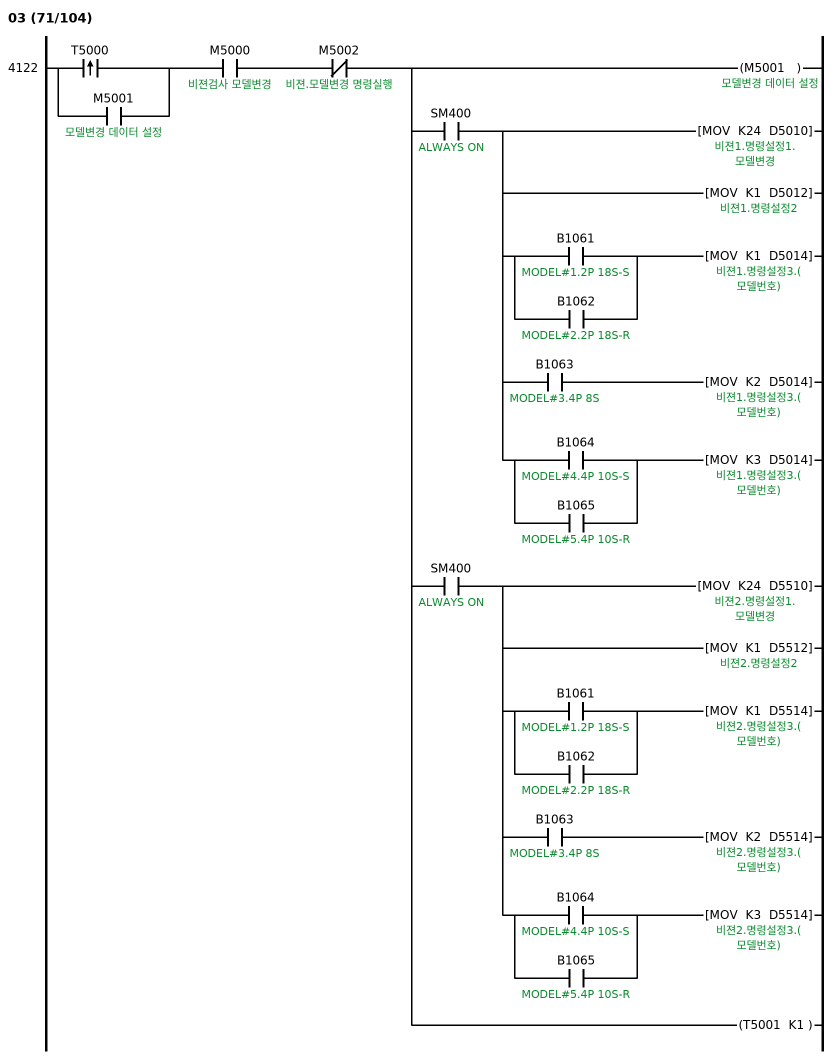
4122  LDP     T5000
      OR      M5001  ; 모델변경 데이터 설정
      AND     M5000  ; 비젼검사 모델변경
      ANI     M5002  ; 비젼.모델변경 명령실행
      OUT     M5001  ; 모델변경 데이터 설정
      MPS
      AND     SM400  ; ALWAYS ON
      MOV     K24 D5010  ; 비젼1.명령설정1.모델변경
      MOV     K1 D5012  ; 비젼1.명령설정2
      MPS
      LD      B1061  ; MODEL#1.2P 18S-S
      OR      B1062  ; MODEL#2.2P 18S-R
      ANB
      MOV     K1 D5014  ; 비젼1.명령설정3.(모델번호)
      MRD
      AND     B1063  ; MODEL#3.4P 8S
      MOV     K2 D5014
      MPP
      LD      B1064  ; MODEL#4.4P 10S-S
      OR      B1065  ; MODEL#5.4P 10S-R
      ANB
      MOV     K3 D5014
      MRD
      AND     SM400  ; ALWAYS ON
      MOV     K24 D5510  ; 비젼2.명령설정1.모델변경
      MOV     K1 D5512  ; 비젼2.명령설정2
      MPS
      LD      B1061  ; MODEL#1.2P 18S-S
      OR      B1062  ; MODEL#2.2P 18S-R
      ANB
      MOV     K1 D5514  ; 비젼2.명령설정3.(모델번호)
      MRD
      AND     B1063  ; MODEL#3.4P 8S
      MOV     K2 D5514
      MPP
      LD      B1064  ; MODEL#4.4P 10S-S
      OR      B1065  ; MODEL#5.4P 10S-R
      ANB
      MOV     K3 D5514
      MPP
      OUT     T5001 K1
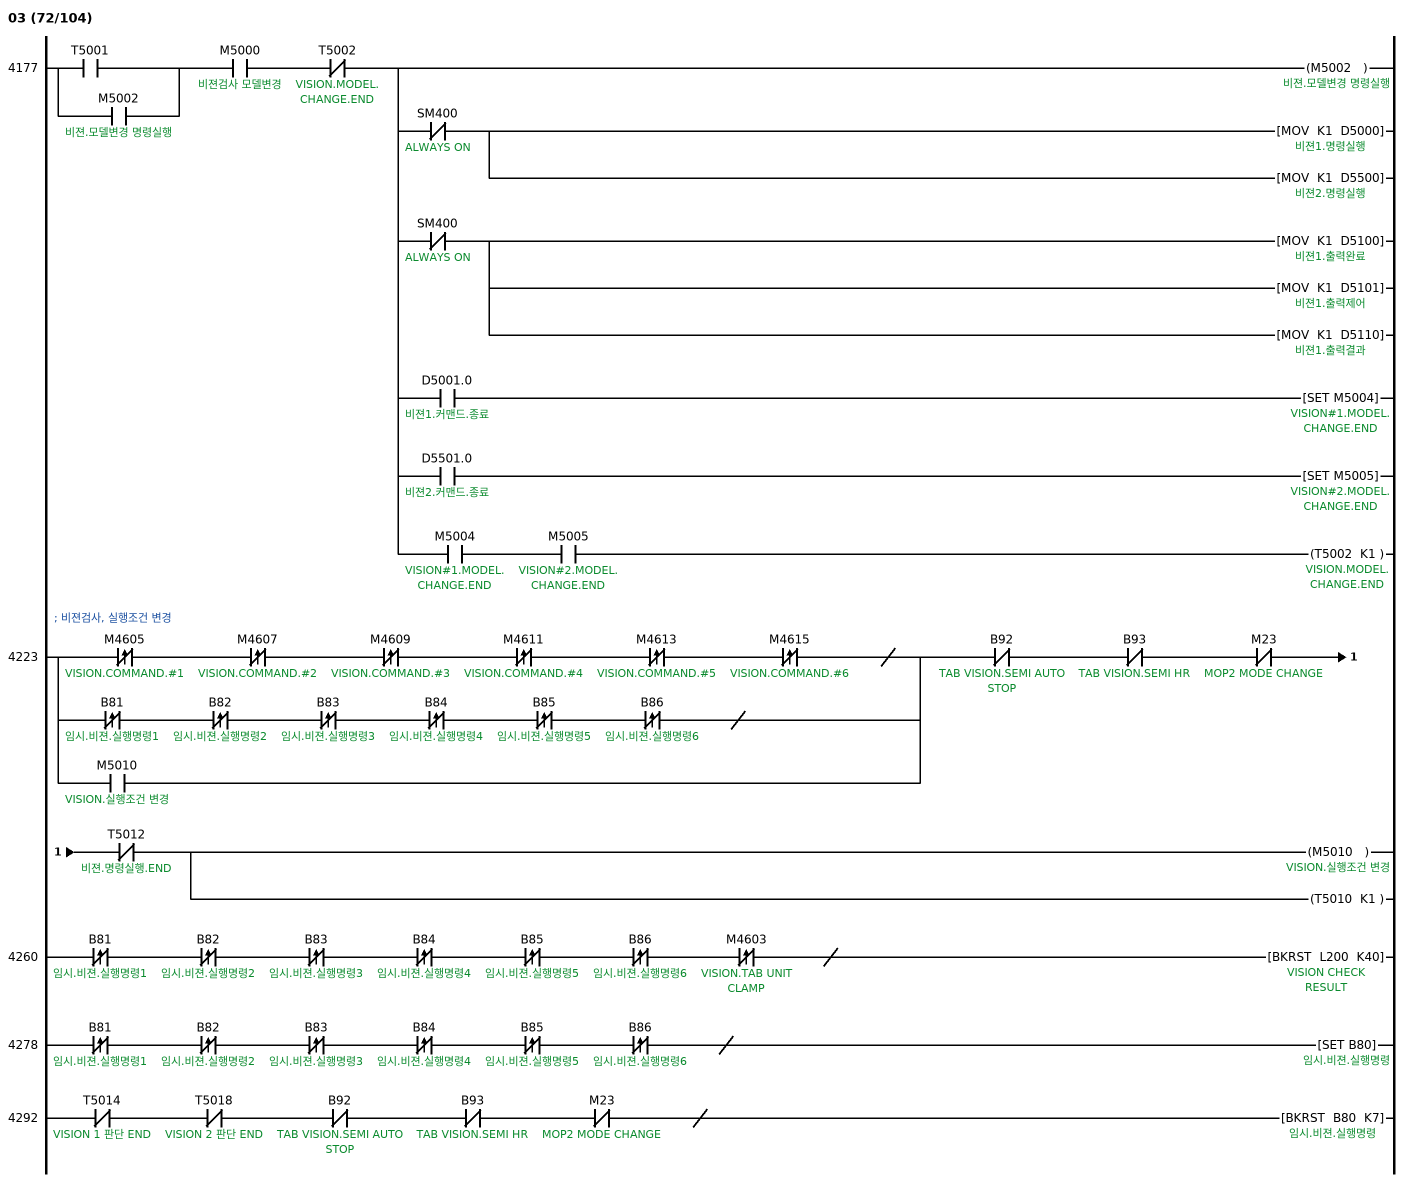
4177  LD      T5001
      OR      M5002  ; 비젼.모델변경 명령실행
      AND     M5000  ; 비젼검사 모델변경
      ANI     T5002  ; VISION.MODEL.CHANGE.END
      OUT     M5002  ; 비젼.모델변경 명령실행
      MPS
      ANI     SM400  ; ALWAYS ON
      MOV     K1 D5000  ; 비젼1.명령실행
      MOV     K1 D5500  ; 비젼2.명령실행
      MRD
      ANI     SM400  ; ALWAYS ON
      MOV     K1 D5100  ; 비젼1.출력완료
      MOV     K1 D5101  ; 비젼1.출력제어
      MOV     K1 D5110  ; 비젼1.출력결과
      MRD
      AND     D5001.0  ; 비젼1.커맨드.종료
      SET     M5004  ; VISION#1.MODEL.CHANGE.END
      MRD
      AND     D5501.0  ; 비젼2.커맨드.종료
      SET     M5005  ; VISION#2.MODEL.CHANGE.END
      MPP
      AND     M5004  ; VISION#1.MODEL.CHANGE.END
      AND     M5005  ; VISION#2.MODEL.CHANGE.END
      OUT     T5002 K1  ; VISION.MODEL.CHANGE.END
; 비젼검사, 실행조건 변경
4223  LDPI    M4605  ; VISION.COMMAND.#1
      ANDPI   M4607  ; VISION.COMMAND.#2
      ANDPI   M4609  ; VISION.COMMAND.#3
      ANDPI   M4611  ; VISION.COMMAND.#4
      ANDPI   M4613  ; VISION.COMMAND.#5
      ANDPI   M4615  ; VISION.COMMAND.#6
      INV
      LDPI    B81  ; 임시.비젼.실행명령1
      ANDPI   B82  ; 임시.비젼.실행명령2
      ANDPI   B83  ; 임시.비젼.실행명령3
      ANDPI   B84  ; 임시.비젼.실행명령4
      ANDPI   B85  ; 임시.비젼.실행명령5
      ANDPI   B86  ; 임시.비젼.실행명령6
      INV
      ORB
      OR      M5010  ; VISION.실행조건 변경
      ANI     B92  ; TAB VISION.SEMI AUTO STOP
      ANI     B93  ; TAB VISION.SEMI HR
      ANI     M23  ; MOP2 MODE CHANGE
      ANI     T5012  ; 비젼.명령실행.END
      OUT     M5010  ; VISION.실행조건 변경
      OUT     T5010 K1
4260  LDPI    B81  ; 임시.비젼.실행명령1
      ANDPI   B82  ; 임시.비젼.실행명령2
      ANDPI   B83  ; 임시.비젼.실행명령3
      ANDPI   B84  ; 임시.비젼.실행명령4
      ANDPI   B85  ; 임시.비젼.실행명령5
      ANDPI   B86  ; 임시.비젼.실행명령6
      ANDPI   M4603  ; VISION.TAB UNIT CLAMP
      INV
      BKRST   L200 K40  ; VISION CHECK RESULT
4278  LDPI    B81  ; 임시.비젼.실행명령1
      ANDPI   B82  ; 임시.비젼.실행명령2
      ANDPI   B83  ; 임시.비젼.실행명령3
      ANDPI   B84  ; 임시.비젼.실행명령4
      ANDPI   B85  ; 임시.비젼.실행명령5
      ANDPI   B86  ; 임시.비젼.실행명령6
      INV
      SET     B80  ; 임시.비젼.실행명령
4292  LDI     T5014  ; VISION 1 판단 END
      ANI     T5018  ; VISION 2 판단 END
      ANI     B92  ; TAB VISION.SEMI AUTO STOP
      ANI     B93  ; TAB VISION.SEMI HR
      ANI     M23  ; MOP2 MODE CHANGE
      INV
      BKRST   B80 K7
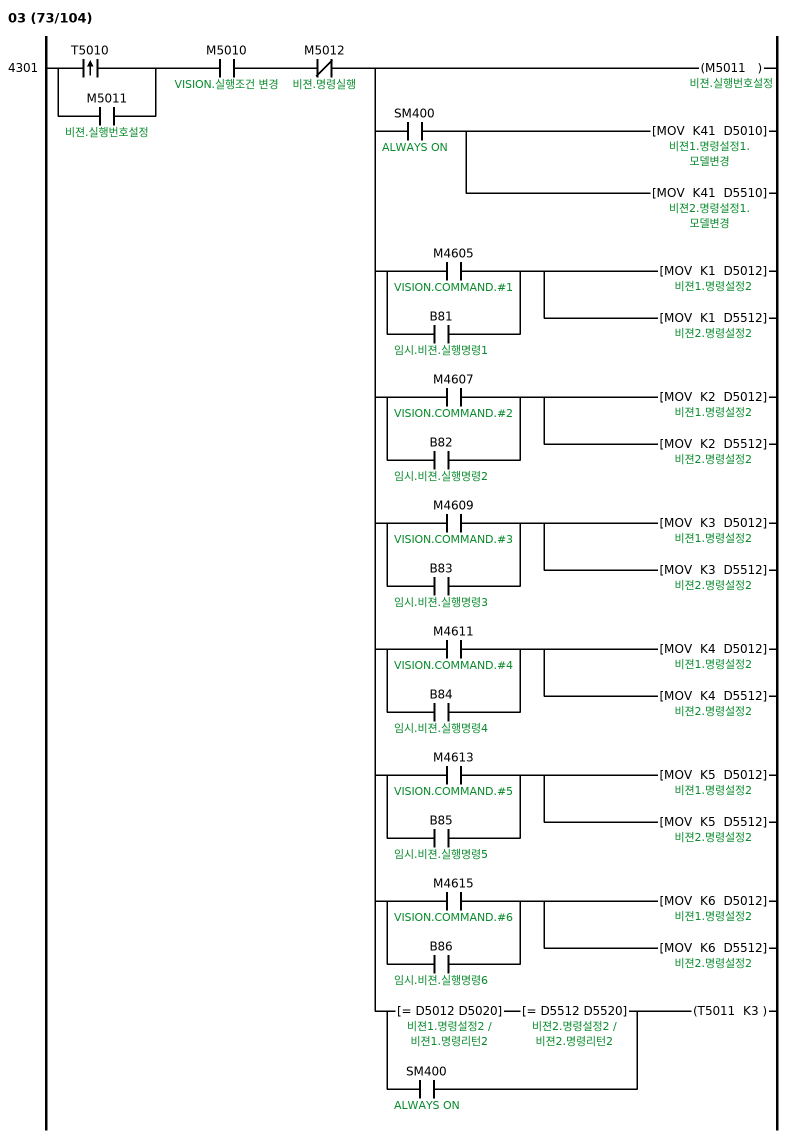
4301  LDP     T5010
      OR      M5011  ; 비젼.실행번호설정
      AND     M5010  ; VISION.실행조건 변경
      ANI     M5012  ; 비젼.명령실행
      OUT     M5011  ; 비젼.실행번호설정
      MPS
      AND     SM400  ; ALWAYS ON
      MOV     K41 D5010
        [note] 실행조건(위치정보)변경
      MOV     K41 D5510
      MRD
      LD      M4605  ; VISION.COMMAND.#1
      OR      B81  ; 임시.비젼.실행명령1
      ANB
      MOV     K1 D5012
        [note] 실행번호(위치번호)설정
      MOV     K1 D5512
      MRD
      LD      M4607  ; VISION.COMMAND.#2
      OR      B82  ; 임시.비젼.실행명령2
      ANB
      MOV     K2 D5012
      MOV     K2 D5512
      MRD
      LD      M4609  ; VISION.COMMAND.#3
      OR      B83  ; 임시.비젼.실행명령3
      ANB
      MOV     K3 D5012
      MOV     K3 D5512
      MRD
      LD      M4611  ; VISION.COMMAND.#4
      OR      B84  ; 임시.비젼.실행명령4
      ANB
      MOV     K4 D5012
      MOV     K4 D5512
      MRD
      LD      M4613  ; VISION.COMMAND.#5
      OR      B85  ; 임시.비젼.실행명령5
      ANB
      MOV     K5 D5012
      MOV     K5 D5512
      MRD
      LD      M4615  ; VISION.COMMAND.#6
      OR      B86  ; 임시.비젼.실행명령6
      ANB
      MOV     K6 D5012
      MOV     K6 D5512
      MPP
      LD=     D5012 D5020  ; 비젼1.명령설정2 / 비젼1.명령리턴2
      AND=    D5512 D5520  ; 비젼2.명령설정2 / 비젼2.명령리턴2
      OR      SM400  ; ALWAYS ON
      ANB
      OUT     T5011 K3
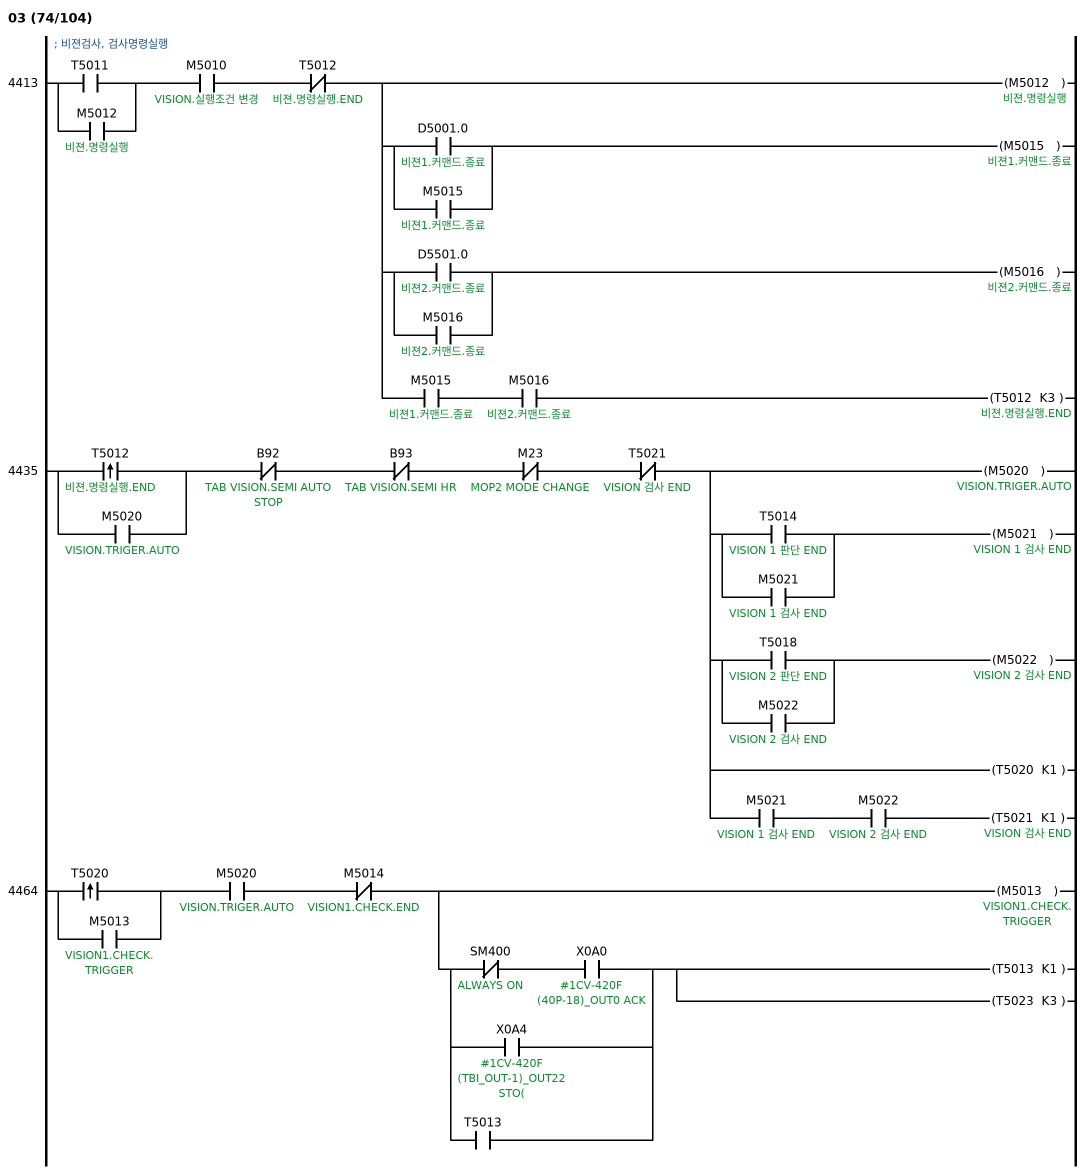
; 비젼검사, 검사명령실행
4413  LD      T5011
      OR      M5012  ; 비젼.명령실행
      AND     M5010  ; VISION.실행조건 변경
      ANI     T5012  ; 비젼.명령실행.END
      OUT     M5012  ; 비젼.명령실행
      MPS
      LD      D5001.0  ; 비젼1.커맨드.종료
      OR      M5015  ; 비젼1.커맨드.종료
      ANB
      OUT     M5015  ; 비젼1.커맨드.종료
      MRD
      LD      D5501.0  ; 비젼2.커맨드.종료
      OR      M5016  ; 비젼2.커맨드.종료
      ANB
      OUT     M5016  ; 비젼2.커맨드.종료
      MPP
      AND     M5015  ; 비젼1.커맨드.종료
      AND     M5016  ; 비젼2.커맨드.종료
      OUT     T5012 K3  ; 비젼.명령실행.END
4435  LDP     T5012  ; 비젼.명령실행.END
      OR      M5020  ; VISION.TRIGER.AUTO
      ANI     B92  ; TAB VISION.SEMI AUTO STOP
      ANI     B93  ; TAB VISION.SEMI HR
      ANI     M23  ; MOP2 MODE CHANGE
      ANI     T5021  ; VISION 검사 END
      OUT     M5020  ; VISION.TRIGER.AUTO
      MPS
      LD      T5014  ; VISION 1 판단 END
      OR      M5021  ; VISION 1 검사 END
      ANB
      OUT     M5021  ; VISION 1 검사 END
      MRD
      LD      T5018  ; VISION 2 판단 END
      OR      M5022  ; VISION 2 검사 END
      ANB
      OUT     M5022  ; VISION 2 검사 END
      MPP
      OUT     T5020 K1
      AND     M5021  ; VISION 1 검사 END
      AND     M5022  ; VISION 2 검사 END
      OUT     T5021 K1  ; VISION 검사 END
4464  LDP     T5020
      OR      M5013  ; VISION1.CHECK.TRIGGER
      AND     M5020  ; VISION.TRIGER.AUTO
      ANI     M5014  ; VISION1.CHECK.END
      OUT     M5013  ; VISION1.CHECK.TRIGGER
      LDI     SM400  ; ALWAYS ON
      AND     X0A0  ; #1CV-420F (40P-18)_OUT0 ACK
      OR      X0A4  ; #1CV-420F (TBI_OUT-1)_OUT22 STO(
      OR      T5013
      ANB
      OUT     T5013 K1
      OUT     T5023 K3
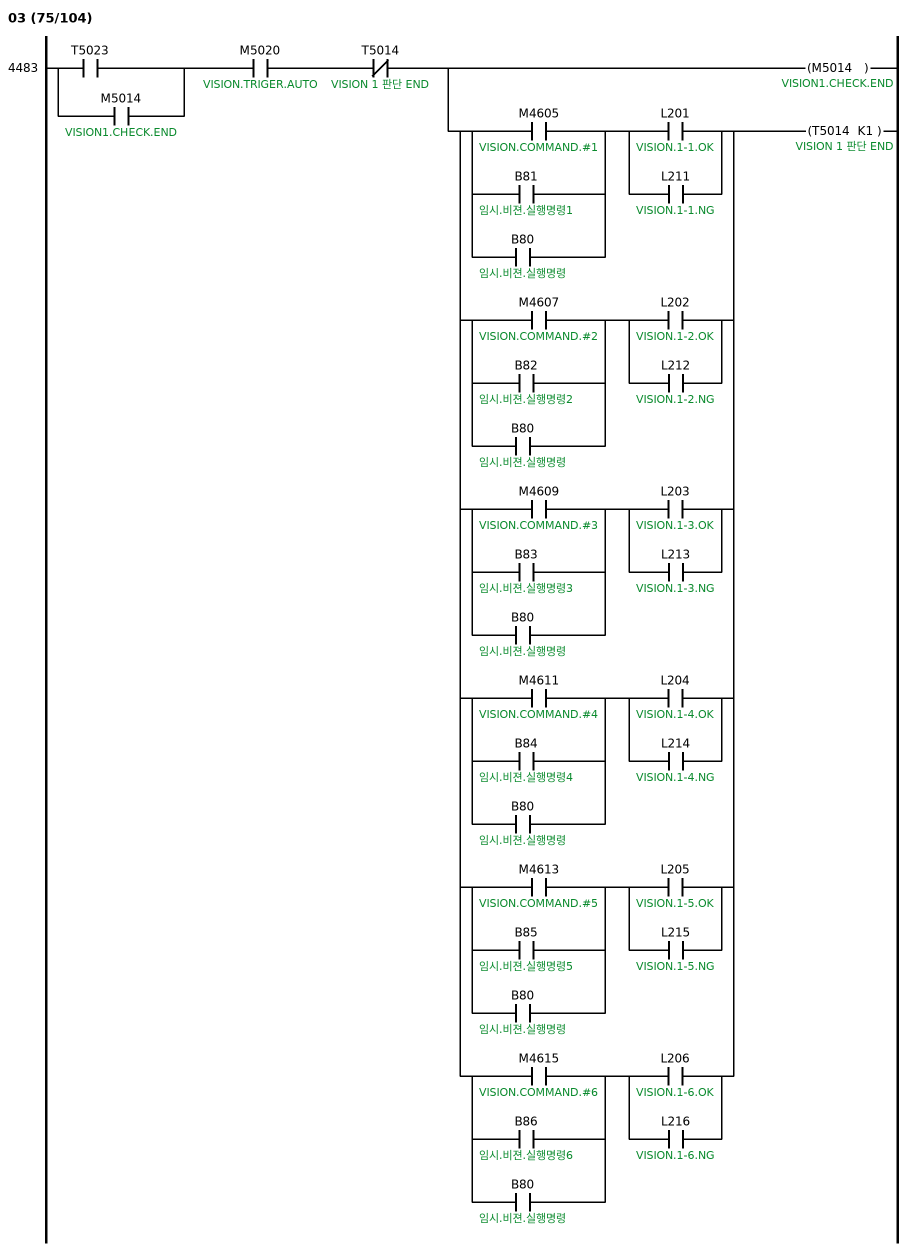
4483  LD      T5023
      OR      M5014  ; VISION1.CHECK.END
      AND     M5020  ; VISION.TRIGER.AUTO
      ANI     T5014  ; VISION 1 판단 END
      OUT     M5014  ; VISION1.CHECK.END
      LD      M4605  ; VISION.COMMAND.#1
      OR      B81  ; 임시.비젼.실행명령1
      OR      B80  ; 임시.비젼.실행명령
      LD      L201  ; VISION.1-1.OK
      OR      L211  ; VISION.1-1.NG
      ANB
      LD      M4607  ; VISION.COMMAND.#2
      OR      B82  ; 임시.비젼.실행명령2
      OR      B80  ; 임시.비젼.실행명령
      LD      L202  ; VISION.1-2.OK
      OR      L212  ; VISION.1-2.NG
      ANB
      ORB
      LD      M4609  ; VISION.COMMAND.#3
      OR      B83  ; 임시.비젼.실행명령3
      OR      B80  ; 임시.비젼.실행명령
      LD      L203  ; VISION.1-3.OK
      OR      L213  ; VISION.1-3.NG
      ANB
      ORB
      LD      M4611  ; VISION.COMMAND.#4
      OR      B84  ; 임시.비젼.실행명령4
      OR      B80  ; 임시.비젼.실행명령
      LD      L204  ; VISION.1-4.OK
      OR      L214  ; VISION.1-4.NG
      ANB
      ORB
      LD      M4613  ; VISION.COMMAND.#5
      OR      B85  ; 임시.비젼.실행명령5
      OR      B80  ; 임시.비젼.실행명령
      LD      L205  ; VISION.1-5.OK
      OR      L215  ; VISION.1-5.NG
      ANB
      ORB
      LD      M4615  ; VISION.COMMAND.#6
      OR      B86  ; 임시.비젼.실행명령6
      OR      B80  ; 임시.비젼.실행명령
      LD      L206  ; VISION.1-6.OK
      OR      L216  ; VISION.1-6.NG
      ANB
      ORB
      ANB
      OUT     T5014 K1  ; VISION 1 판단 END
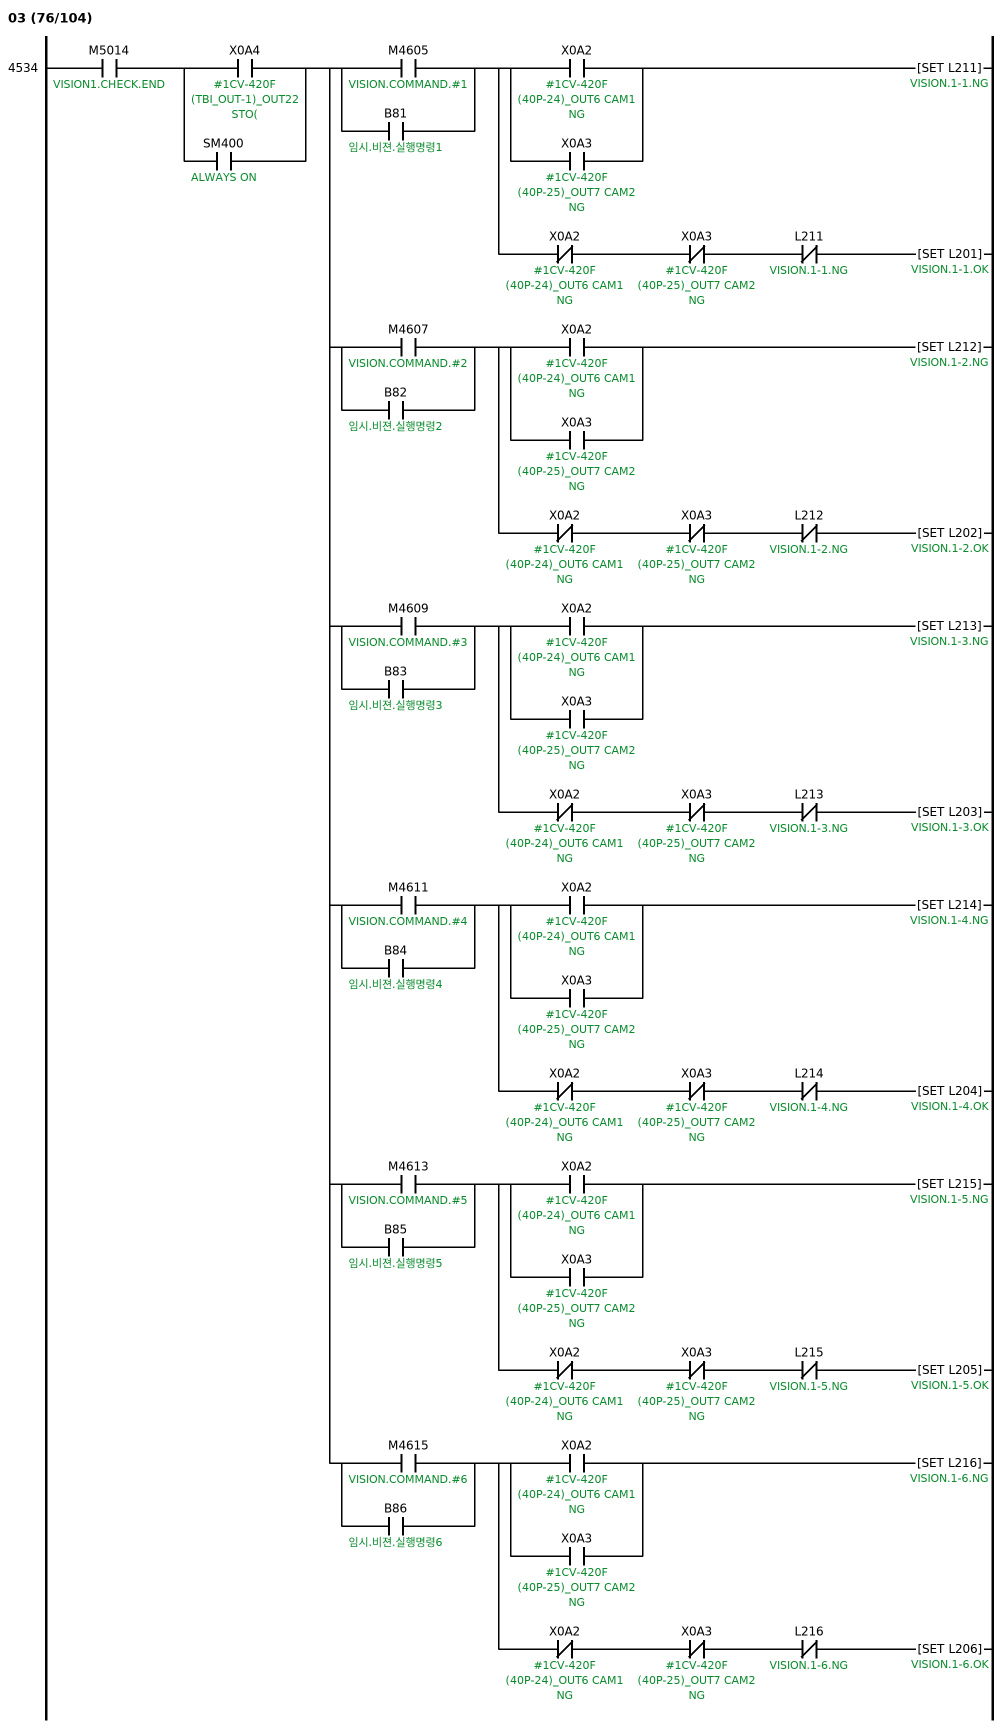
4534  LD      M5014  ; VISION1.CHECK.END
      LD      X0A4  ; #1CV-420F (TBI_OUT-1)_OUT22 STO(
      OR      SM400  ; ALWAYS ON
      ANB
      MPS
      LD      M4605  ; VISION.COMMAND.#1
      OR      B81  ; 임시.비젼.실행명령1
      ANB
      MPS
      LD      X0A2  ; #1CV-420F (40P-24)_OUT6 CAM1 NG
      OR      X0A3  ; #1CV-420F (40P-25)_OUT7 CAM2 NG
      ANB
      SET     L211  ; VISION.1-1.NG
      MPP
      ANI     X0A2  ; #1CV-420F (40P-24)_OUT6 CAM1 NG
      ANI     X0A3  ; #1CV-420F (40P-25)_OUT7 CAM2 NG
      ANI     L211  ; VISION.1-1.NG
      SET     L201  ; VISION.1-1.OK
      MRD
      LD      M4607  ; VISION.COMMAND.#2
      OR      B82  ; 임시.비젼.실행명령2
      ANB
      MPS
      LD      X0A2  ; #1CV-420F (40P-24)_OUT6 CAM1 NG
      OR      X0A3  ; #1CV-420F (40P-25)_OUT7 CAM2 NG
      ANB
      SET     L212  ; VISION.1-2.NG
      MPP
      ANI     X0A2  ; #1CV-420F (40P-24)_OUT6 CAM1 NG
      ANI     X0A3  ; #1CV-420F (40P-25)_OUT7 CAM2 NG
      ANI     L212  ; VISION.1-2.NG
      SET     L202  ; VISION.1-2.OK
      MRD
      LD      M4609  ; VISION.COMMAND.#3
      OR      B83  ; 임시.비젼.실행명령3
      ANB
      MPS
      LD      X0A2  ; #1CV-420F (40P-24)_OUT6 CAM1 NG
      OR      X0A3  ; #1CV-420F (40P-25)_OUT7 CAM2 NG
      ANB
      SET     L213  ; VISION.1-3.NG
      MPP
      ANI     X0A2  ; #1CV-420F (40P-24)_OUT6 CAM1 NG
      ANI     X0A3  ; #1CV-420F (40P-25)_OUT7 CAM2 NG
      ANI     L213  ; VISION.1-3.NG
      SET     L203  ; VISION.1-3.OK
      MRD
      LD      M4611  ; VISION.COMMAND.#4
      OR      B84  ; 임시.비젼.실행명령4
      ANB
      MPS
      LD      X0A2  ; #1CV-420F (40P-24)_OUT6 CAM1 NG
      OR      X0A3  ; #1CV-420F (40P-25)_OUT7 CAM2 NG
      ANB
      SET     L214  ; VISION.1-4.NG
      MPP
      ANI     X0A2  ; #1CV-420F (40P-24)_OUT6 CAM1 NG
      ANI     X0A3  ; #1CV-420F (40P-25)_OUT7 CAM2 NG
      ANI     L214  ; VISION.1-4.NG
      SET     L204  ; VISION.1-4.OK
      MRD
      LD      M4613  ; VISION.COMMAND.#5
      OR      B85  ; 임시.비젼.실행명령5
      ANB
      MPS
      LD      X0A2  ; #1CV-420F (40P-24)_OUT6 CAM1 NG
      OR      X0A3  ; #1CV-420F (40P-25)_OUT7 CAM2 NG
      ANB
      SET     L215  ; VISION.1-5.NG
      MPP
      ANI     X0A2  ; #1CV-420F (40P-24)_OUT6 CAM1 NG
      ANI     X0A3  ; #1CV-420F (40P-25)_OUT7 CAM2 NG
      ANI     L215  ; VISION.1-5.NG
      SET     L205  ; VISION.1-5.OK
      MPP
      LD      M4615  ; VISION.COMMAND.#6
      OR      B86  ; 임시.비젼.실행명령6
      ANB
      MPS
      LD      X0A2  ; #1CV-420F (40P-24)_OUT6 CAM1 NG
      OR      X0A3  ; #1CV-420F (40P-25)_OUT7 CAM2 NG
      ANB
      SET     L216  ; VISION.1-6.NG
      MPP
      ANI     X0A2  ; #1CV-420F (40P-24)_OUT6 CAM1 NG
      ANI     X0A3  ; #1CV-420F (40P-25)_OUT7 CAM2 NG
      ANI     L216  ; VISION.1-6.NG
      SET     L206  ; VISION.1-6.OK
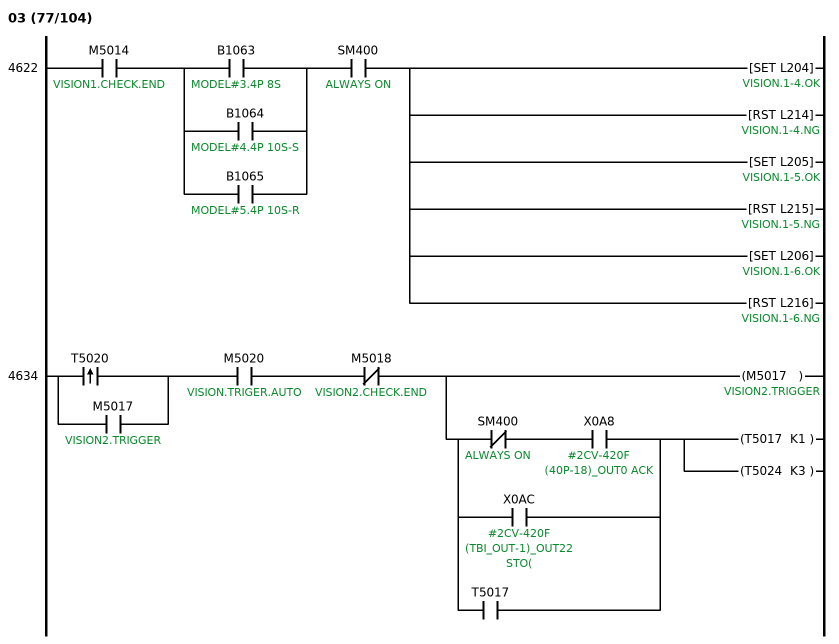
4622  LD      M5014  ; VISION1.CHECK.END
      LD      B1063  ; MODEL#3.4P 8S
      OR      B1064  ; MODEL#4.4P 10S-S
      OR      B1065  ; MODEL#5.4P 10S-R
      ANB
      AND     SM400  ; ALWAYS ON
      SET     L204  ; VISION.1-4.OK
      RST     L214  ; VISION.1-4.NG
      SET     L205  ; VISION.1-5.OK
      RST     L215  ; VISION.1-5.NG
      SET     L206  ; VISION.1-6.OK
      RST     L216  ; VISION.1-6.NG
4634  LDP     T5020
      OR      M5017  ; VISION2.TRIGGER
      AND     M5020  ; VISION.TRIGER.AUTO
      ANI     M5018  ; VISION2.CHECK.END
      OUT     M5017  ; VISION2.TRIGGER
      LDI     SM400  ; ALWAYS ON
      AND     X0A8  ; #2CV-420F (40P-18)_OUT0 ACK
      OR      X0AC  ; #2CV-420F (TBI_OUT-1)_OUT22 STO(
      OR      T5017
      ANB
      OUT     T5017 K1
      OUT     T5024 K3
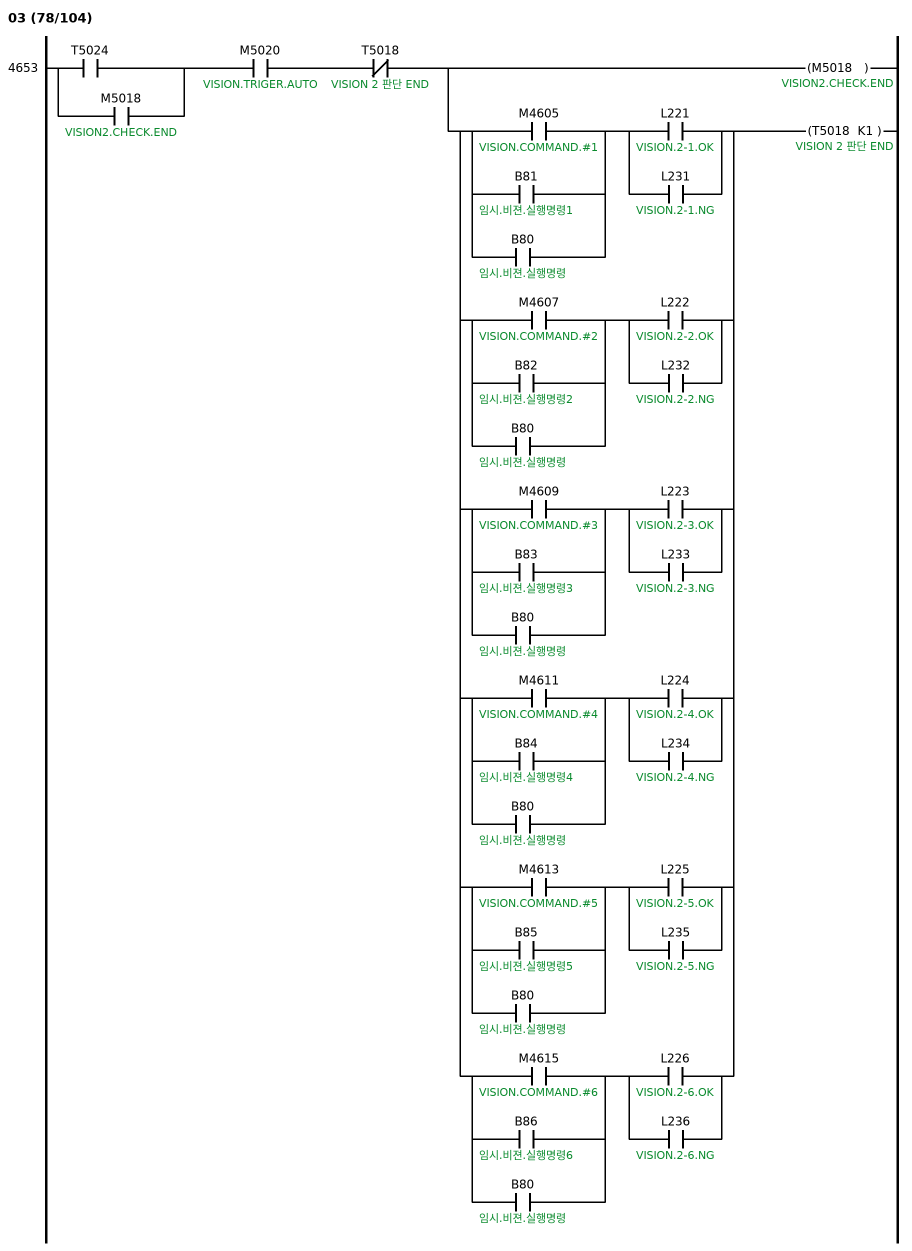
4653  LD      T5024
      OR      M5018  ; VISION2.CHECK.END
      AND     M5020  ; VISION.TRIGER.AUTO
      ANI     T5018  ; VISION 2 판단 END
      OUT     M5018  ; VISION2.CHECK.END
      LD      M4605  ; VISION.COMMAND.#1
      OR      B81  ; 임시.비젼.실행명령1
      OR      B80  ; 임시.비젼.실행명령
      LD      L221  ; VISION.2-1.OK
      OR      L231  ; VISION.2-1.NG
      ANB
      LD      M4607  ; VISION.COMMAND.#2
      OR      B82  ; 임시.비젼.실행명령2
      OR      B80  ; 임시.비젼.실행명령
      LD      L222  ; VISION.2-2.OK
      OR      L232  ; VISION.2-2.NG
      ANB
      ORB
      LD      M4609  ; VISION.COMMAND.#3
      OR      B83  ; 임시.비젼.실행명령3
      OR      B80  ; 임시.비젼.실행명령
      LD      L223  ; VISION.2-3.OK
      OR      L233  ; VISION.2-3.NG
      ANB
      ORB
      LD      M4611  ; VISION.COMMAND.#4
      OR      B84  ; 임시.비젼.실행명령4
      OR      B80  ; 임시.비젼.실행명령
      LD      L224  ; VISION.2-4.OK
      OR      L234  ; VISION.2-4.NG
      ANB
      ORB
      LD      M4613  ; VISION.COMMAND.#5
      OR      B85  ; 임시.비젼.실행명령5
      OR      B80  ; 임시.비젼.실행명령
      LD      L225  ; VISION.2-5.OK
      OR      L235  ; VISION.2-5.NG
      ANB
      ORB
      LD      M4615  ; VISION.COMMAND.#6
      OR      B86  ; 임시.비젼.실행명령6
      OR      B80  ; 임시.비젼.실행명령
      LD      L226  ; VISION.2-6.OK
      OR      L236  ; VISION.2-6.NG
      ANB
      ORB
      ANB
      OUT     T5018 K1  ; VISION 2 판단 END
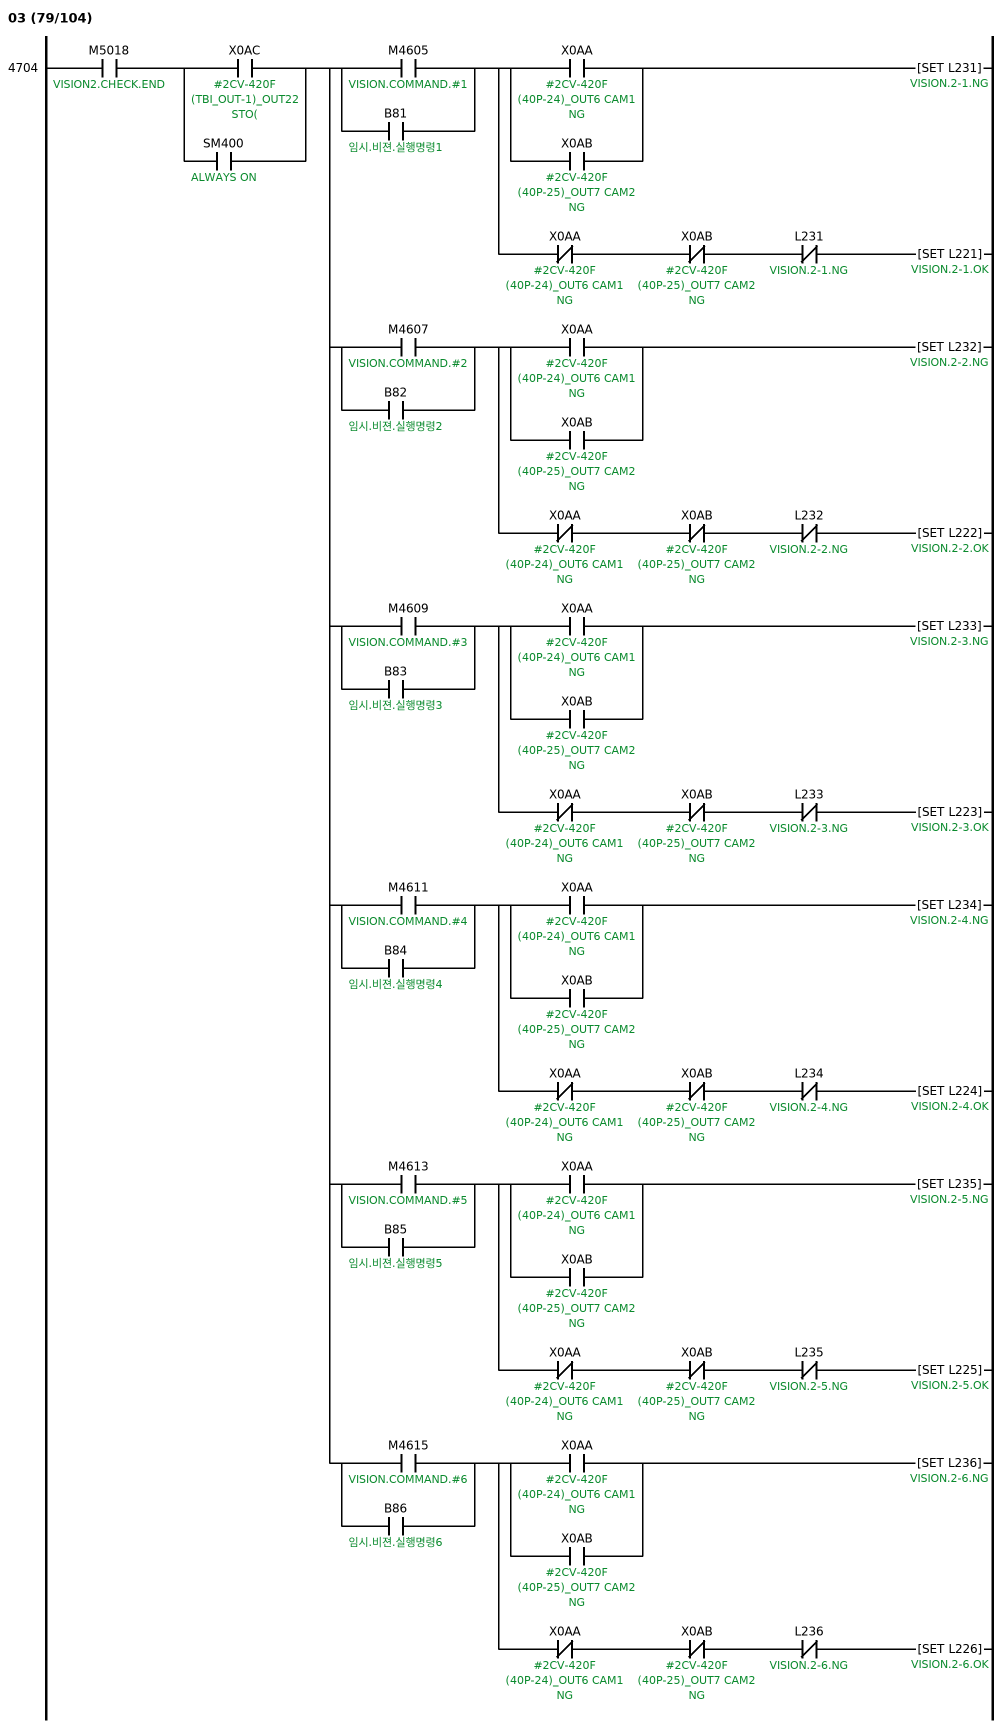
4704  LD      M5018  ; VISION2.CHECK.END
      LD      X0AC  ; #2CV-420F (TBI_OUT-1)_OUT22 STO(
      OR      SM400  ; ALWAYS ON
      ANB
      MPS
      LD      M4605  ; VISION.COMMAND.#1
      OR      B81  ; 임시.비젼.실행명령1
      ANB
      MPS
      LD      X0AA  ; #2CV-420F (40P-24)_OUT6 CAM1 NG
      OR      X0AB  ; #2CV-420F (40P-25)_OUT7 CAM2 NG
      ANB
      SET     L231  ; VISION.2-1.NG
      MPP
      ANI     X0AA  ; #2CV-420F (40P-24)_OUT6 CAM1 NG
      ANI     X0AB  ; #2CV-420F (40P-25)_OUT7 CAM2 NG
      ANI     L231  ; VISION.2-1.NG
      SET     L221  ; VISION.2-1.OK
      MRD
      LD      M4607  ; VISION.COMMAND.#2
      OR      B82  ; 임시.비젼.실행명령2
      ANB
      MPS
      LD      X0AA  ; #2CV-420F (40P-24)_OUT6 CAM1 NG
      OR      X0AB  ; #2CV-420F (40P-25)_OUT7 CAM2 NG
      ANB
      SET     L232  ; VISION.2-2.NG
      MPP
      ANI     X0AA  ; #2CV-420F (40P-24)_OUT6 CAM1 NG
      ANI     X0AB  ; #2CV-420F (40P-25)_OUT7 CAM2 NG
      ANI     L232  ; VISION.2-2.NG
      SET     L222  ; VISION.2-2.OK
      MRD
      LD      M4609  ; VISION.COMMAND.#3
      OR      B83  ; 임시.비젼.실행명령3
      ANB
      MPS
      LD      X0AA  ; #2CV-420F (40P-24)_OUT6 CAM1 NG
      OR      X0AB  ; #2CV-420F (40P-25)_OUT7 CAM2 NG
      ANB
      SET     L233  ; VISION.2-3.NG
      MPP
      ANI     X0AA  ; #2CV-420F (40P-24)_OUT6 CAM1 NG
      ANI     X0AB  ; #2CV-420F (40P-25)_OUT7 CAM2 NG
      ANI     L233  ; VISION.2-3.NG
      SET     L223  ; VISION.2-3.OK
      MRD
      LD      M4611  ; VISION.COMMAND.#4
      OR      B84  ; 임시.비젼.실행명령4
      ANB
      MPS
      LD      X0AA  ; #2CV-420F (40P-24)_OUT6 CAM1 NG
      OR      X0AB  ; #2CV-420F (40P-25)_OUT7 CAM2 NG
      ANB
      SET     L234  ; VISION.2-4.NG
      MPP
      ANI     X0AA  ; #2CV-420F (40P-24)_OUT6 CAM1 NG
      ANI     X0AB  ; #2CV-420F (40P-25)_OUT7 CAM2 NG
      ANI     L234  ; VISION.2-4.NG
      SET     L224  ; VISION.2-4.OK
      MRD
      LD      M4613  ; VISION.COMMAND.#5
      OR      B85  ; 임시.비젼.실행명령5
      ANB
      MPS
      LD      X0AA  ; #2CV-420F (40P-24)_OUT6 CAM1 NG
      OR      X0AB  ; #2CV-420F (40P-25)_OUT7 CAM2 NG
      ANB
      SET     L235  ; VISION.2-5.NG
      MPP
      ANI     X0AA  ; #2CV-420F (40P-24)_OUT6 CAM1 NG
      ANI     X0AB  ; #2CV-420F (40P-25)_OUT7 CAM2 NG
      ANI     L235  ; VISION.2-5.NG
      SET     L225  ; VISION.2-5.OK
      MPP
      LD      M4615  ; VISION.COMMAND.#6
      OR      B86  ; 임시.비젼.실행명령6
      ANB
      MPS
      LD      X0AA  ; #2CV-420F (40P-24)_OUT6 CAM1 NG
      OR      X0AB  ; #2CV-420F (40P-25)_OUT7 CAM2 NG
      ANB
      SET     L236  ; VISION.2-6.NG
      MPP
      ANI     X0AA  ; #2CV-420F (40P-24)_OUT6 CAM1 NG
      ANI     X0AB  ; #2CV-420F (40P-25)_OUT7 CAM2 NG
      ANI     L236  ; VISION.2-6.NG
      SET     L226  ; VISION.2-6.OK
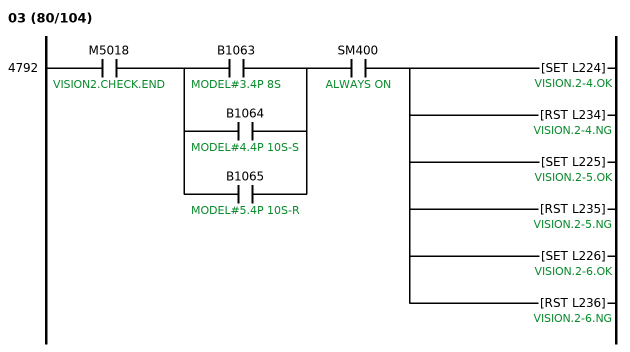
4792  LD      M5018  ; VISION2.CHECK.END
      LD      B1063  ; MODEL#3.4P 8S
      OR      B1064  ; MODEL#4.4P 10S-S
      OR      B1065  ; MODEL#5.4P 10S-R
      ANB
      AND     SM400  ; ALWAYS ON
      SET     L224  ; VISION.2-4.OK
      RST     L234  ; VISION.2-4.NG
      SET     L225  ; VISION.2-5.OK
      RST     L235  ; VISION.2-5.NG
      SET     L226  ; VISION.2-6.OK
      RST     L236  ; VISION.2-6.NG
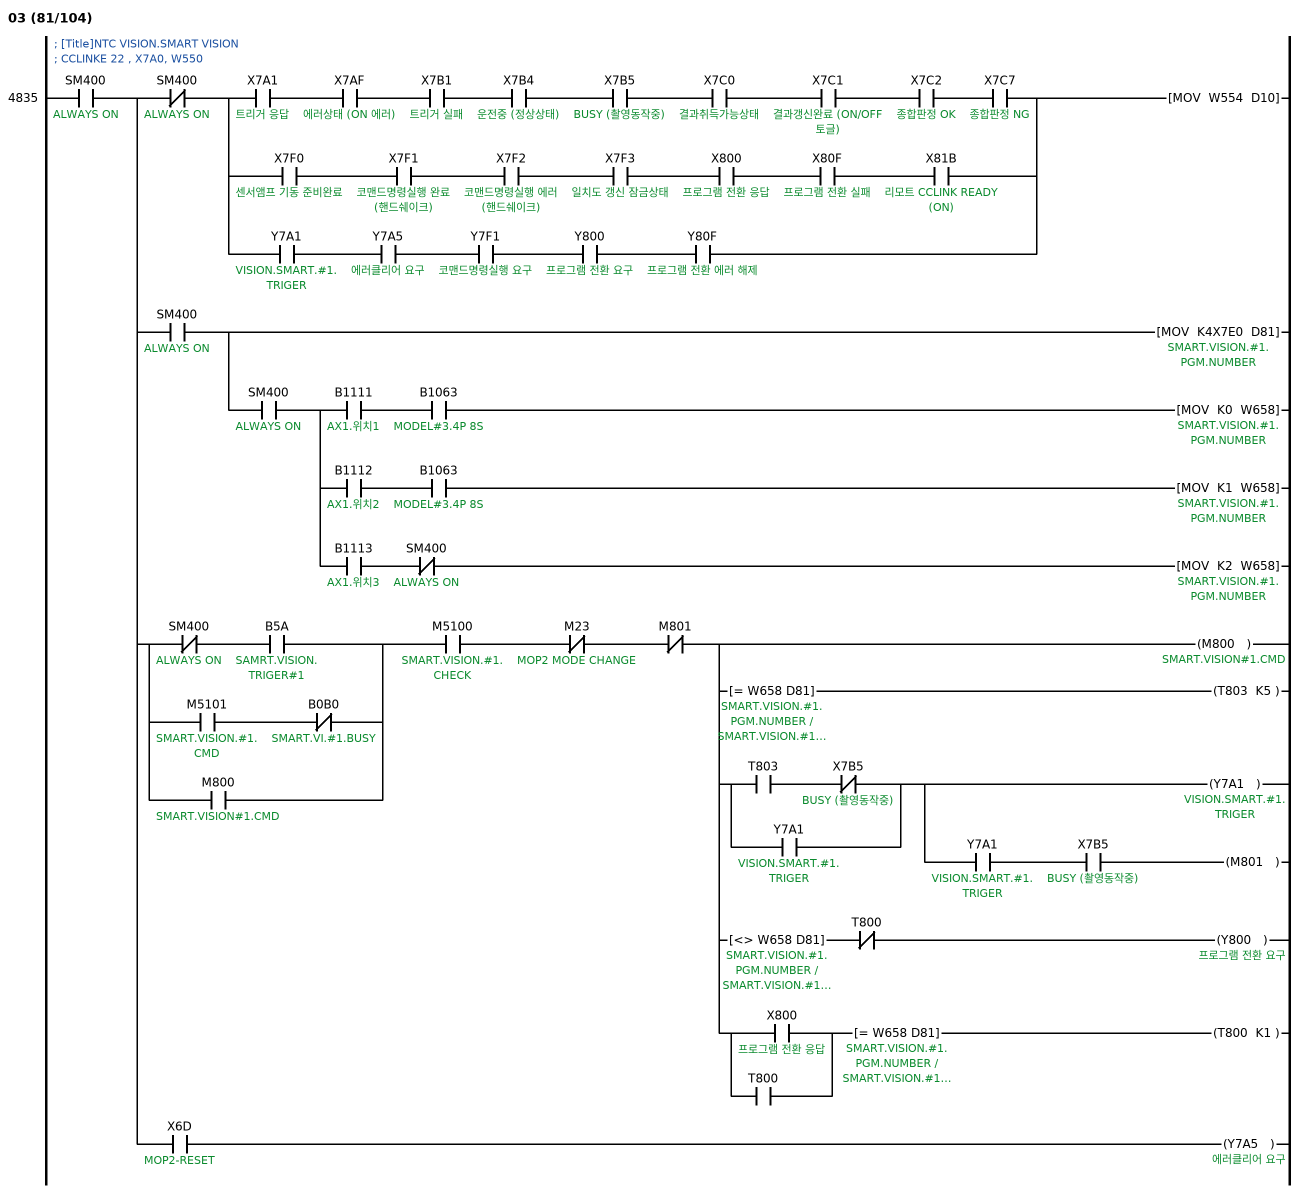
; [Title]NTC VISION.SMART VISION
; CCLINKE 22 , X7A0, W550
4835  LD      SM400  ; ALWAYS ON
      MPS
      ANI     SM400  ; ALWAYS ON
      LD      X7A1  ; 트리거 응답
      AND     X7AF  ; 에러상태 (ON 에러)
      AND     X7B1  ; 트리거 실패
      AND     X7B4  ; 운전중 (정상상태)
      AND     X7B5  ; BUSY (촬영동작중)
      AND     X7C0  ; 결과취득가능상태
      AND     X7C1  ; 결과갱신완료 (ON/OFF 토글)
      AND     X7C2  ; 종합판정 OK
      AND     X7C7  ; 종합판정 NG
      LD      X7F0  ; 센서앰프 기동 준비완료
      AND     X7F1  ; 코맨드명령실행 완료 (핸드쉐이크)
      AND     X7F2  ; 코맨드명령실행 에러 (핸드쉐이크)
      AND     X7F3  ; 일치도 갱신 잠금상태
      AND     X800  ; 프로그램 전환 응답
      AND     X80F  ; 프로그램 전환 실패
      AND     X81B  ; 리모트 CCLINK READY (ON)
      ORB
      LD      Y7A1  ; VISION.SMART.#1.TRIGER
      AND     Y7A5  ; 에러클리어 요구
      AND     Y7F1  ; 코맨드명령실행 요구
      AND     Y800  ; 프로그램 전환 요구
      AND     Y80F  ; 프로그램 전환 에러 해제
      ORB
      ANB
      MOV     W554 D10
      MRD
      AND     SM400  ; ALWAYS ON
      MOV     K4X7E0 D81  ; 프로그램번호 (BIT 0) / SMART.VISION.#1.PGM.NUMBER
      AND     SM400  ; ALWAYS ON
      MPS
      AND     B1111  ; AX1.위치1
      AND     B1063  ; MODEL#3.4P 8S
      MOV     K0 W658  ; SMART.VISION.#1.PGM.NUMBER
      MRD
      AND     B1112  ; AX1.위치2
      AND     B1063  ; MODEL#3.4P 8S
      MOV     K1 W658
      MPP
      AND     B1113  ; AX1.위치3
      ANI     SM400  ; ALWAYS ON
      MOV     K2 W658
      MRD
      LDI     SM400  ; ALWAYS ON
      AND     B5A  ; SAMRT.VISION.TRIGER#1
      LD      M5101  ; SMART.VISION.#1.CMD
      ANI     B0B0  ; SMART.VI.#1.BUSY
      ORB
      OR      M800  ; SMART.VISION#1.CMD
      ANB
      AND     M5100  ; SMART.VISION.#1.CHECK
      ANI     M23  ; MOP2 MODE CHANGE
      ANI     M801
      OUT     M800  ; SMART.VISION#1.CMD
      MPS
      AND=    W658 D81  ; SMART.VISION.#1.PGM.NUMBER / SMART.VISION.#1.PGM.NUMBER
      OUT     T803 K5
      MRD
      LD      T803
      ANI     X7B5  ; BUSY (촬영동작중)
      OR      Y7A1  ; VISION.SMART.#1.TRIGER
      ANB
      OUT     Y7A1  ; VISION.SMART.#1.TRIGER
      AND     Y7A1  ; VISION.SMART.#1.TRIGER
      AND     X7B5  ; BUSY (촬영동작중)
      OUT     M801
      MRD
      AND<>   W658 D81  ; SMART.VISION.#1.PGM.NUMBER / SMART.VISION.#1.PGM.NUMBER
      ANI     T800
      OUT     Y800  ; 프로그램 전환 요구
      MPP
      LD      X800  ; 프로그램 전환 응답
      OR      T800
      ANB
      AND=    W658 D81  ; SMART.VISION.#1.PGM.NUMBER / SMART.VISION.#1.PGM.NUMBER
      OUT     T800 K1
      MPP
      AND     X6D  ; MOP2-RESET
      OUT     Y7A5  ; 에러클리어 요구
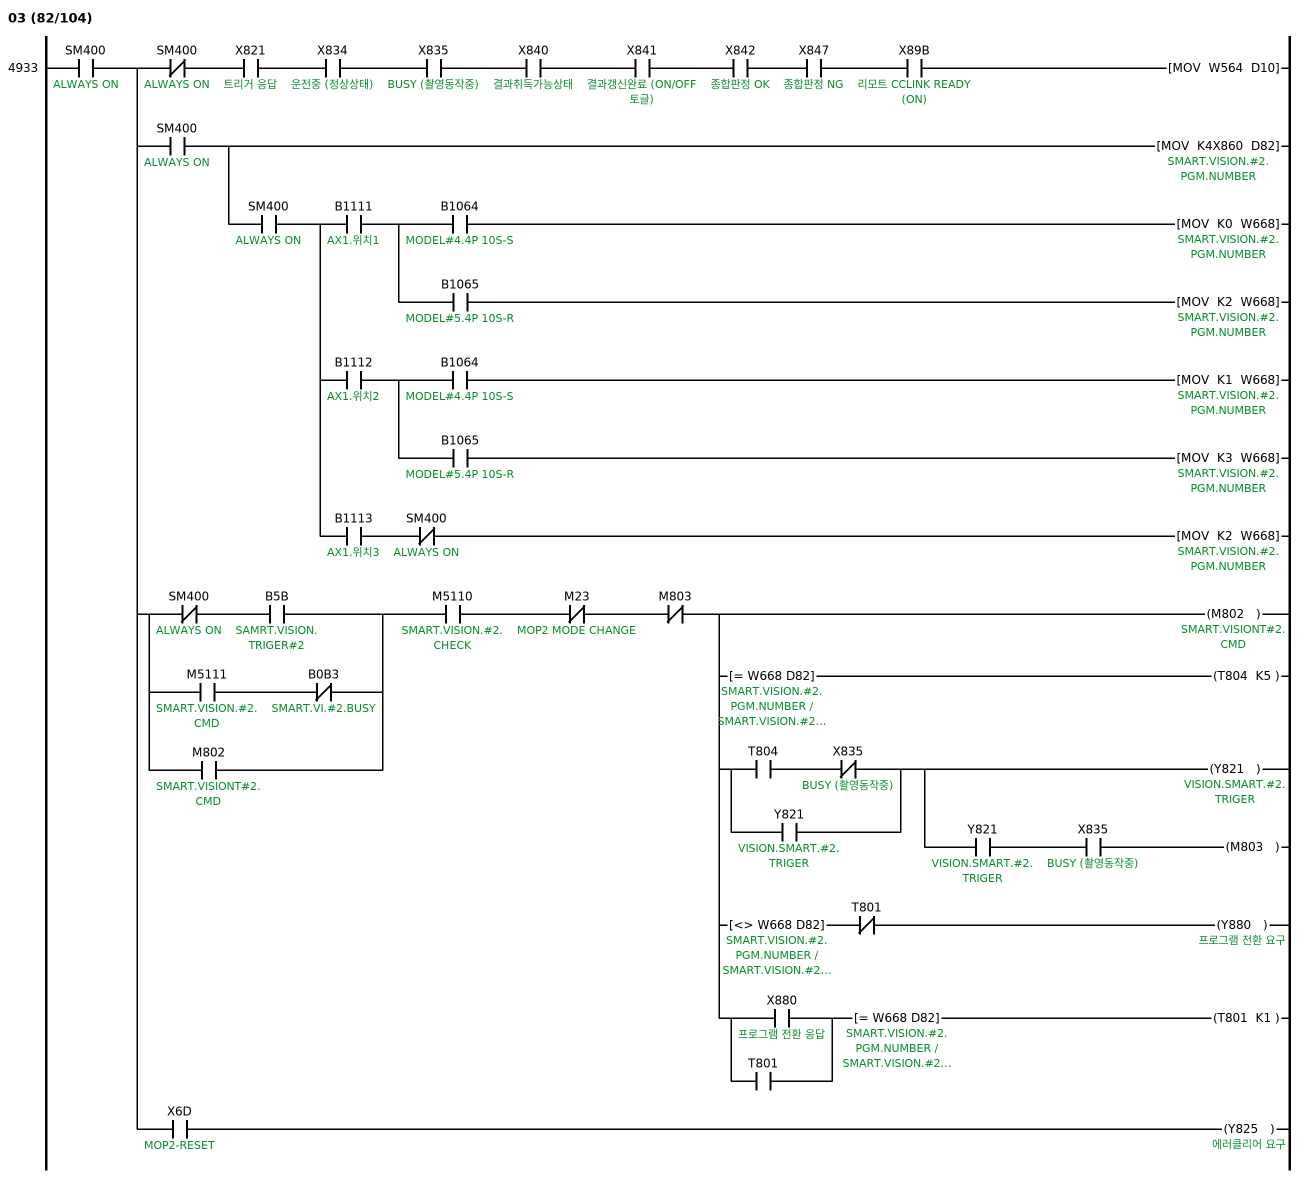
4933  LD      SM400  ; ALWAYS ON
      MPS
      ANI     SM400  ; ALWAYS ON
      AND     X821  ; 트리거 응답
      AND     X834  ; 운전중 (정상상태)
      AND     X835  ; BUSY (촬영동작중)
      AND     X840  ; 결과취득가능상태
      AND     X841  ; 결과갱신완료 (ON/OFF 토글)
      AND     X842  ; 종합판정 OK
      AND     X847  ; 종합판정 NG
      AND     X89B  ; 리모트 CCLINK READY (ON)
      MOV     W564 D10
      MRD
      AND     SM400  ; ALWAYS ON
      MOV     K4X860 D82  ; 프로그램번호 (BIT 0) / SMART.VISION.#2.PGM.NUMBER
      AND     SM400  ; ALWAYS ON
      MPS
      AND     B1111  ; AX1.위치1
      MPS
      AND     B1064  ; MODEL#4.4P 10S-S
      MOV     K0 W668  ; SMART.VISION.#2.PGM.NUMBER
      MPP
      AND     B1065  ; MODEL#5.4P 10S-R
      MOV     K2 W668
      MRD
      AND     B1112  ; AX1.위치2
      MPS
      AND     B1064  ; MODEL#4.4P 10S-S
      MOV     K1 W668
      MPP
      AND     B1065  ; MODEL#5.4P 10S-R
      MOV     K3 W668
      MPP
      AND     B1113  ; AX1.위치3
      ANI     SM400  ; ALWAYS ON
      MOV     K2 W668
      MRD
      LDI     SM400  ; ALWAYS ON
      AND     B5B  ; SAMRT.VISION.TRIGER#2
      LD      M5111  ; SMART.VISION.#2.CMD
      ANI     B0B3  ; SMART.VI.#2.BUSY
      ORB
      OR      M802  ; SMART.VISIONT#2.CMD
      ANB
      AND     M5110  ; SMART.VISION.#2.CHECK
      ANI     M23  ; MOP2 MODE CHANGE
      ANI     M803
      OUT     M802  ; SMART.VISIONT#2.CMD
      MPS
      AND=    W668 D82  ; SMART.VISION.#2.PGM.NUMBER / SMART.VISION.#2.PGM.NUMBER
      OUT     T804 K5
      MRD
      LD      T804
      ANI     X835  ; BUSY (촬영동작중)
      OR      Y821  ; VISION.SMART.#2.TRIGER
      ANB
      OUT     Y821  ; VISION.SMART.#2.TRIGER
      AND     Y821  ; VISION.SMART.#2.TRIGER
      AND     X835  ; BUSY (촬영동작중)
      OUT     M803
      MRD
      AND<>   W668 D82  ; SMART.VISION.#2.PGM.NUMBER / SMART.VISION.#2.PGM.NUMBER
      ANI     T801
      OUT     Y880  ; 프로그램 전환 요구
      MPP
      LD      X880  ; 프로그램 전환 응답
      OR      T801
      ANB
      AND=    W668 D82  ; SMART.VISION.#2.PGM.NUMBER / SMART.VISION.#2.PGM.NUMBER
      OUT     T801 K1
      MPP
      AND     X6D  ; MOP2-RESET
      OUT     Y825  ; 에러클리어 요구
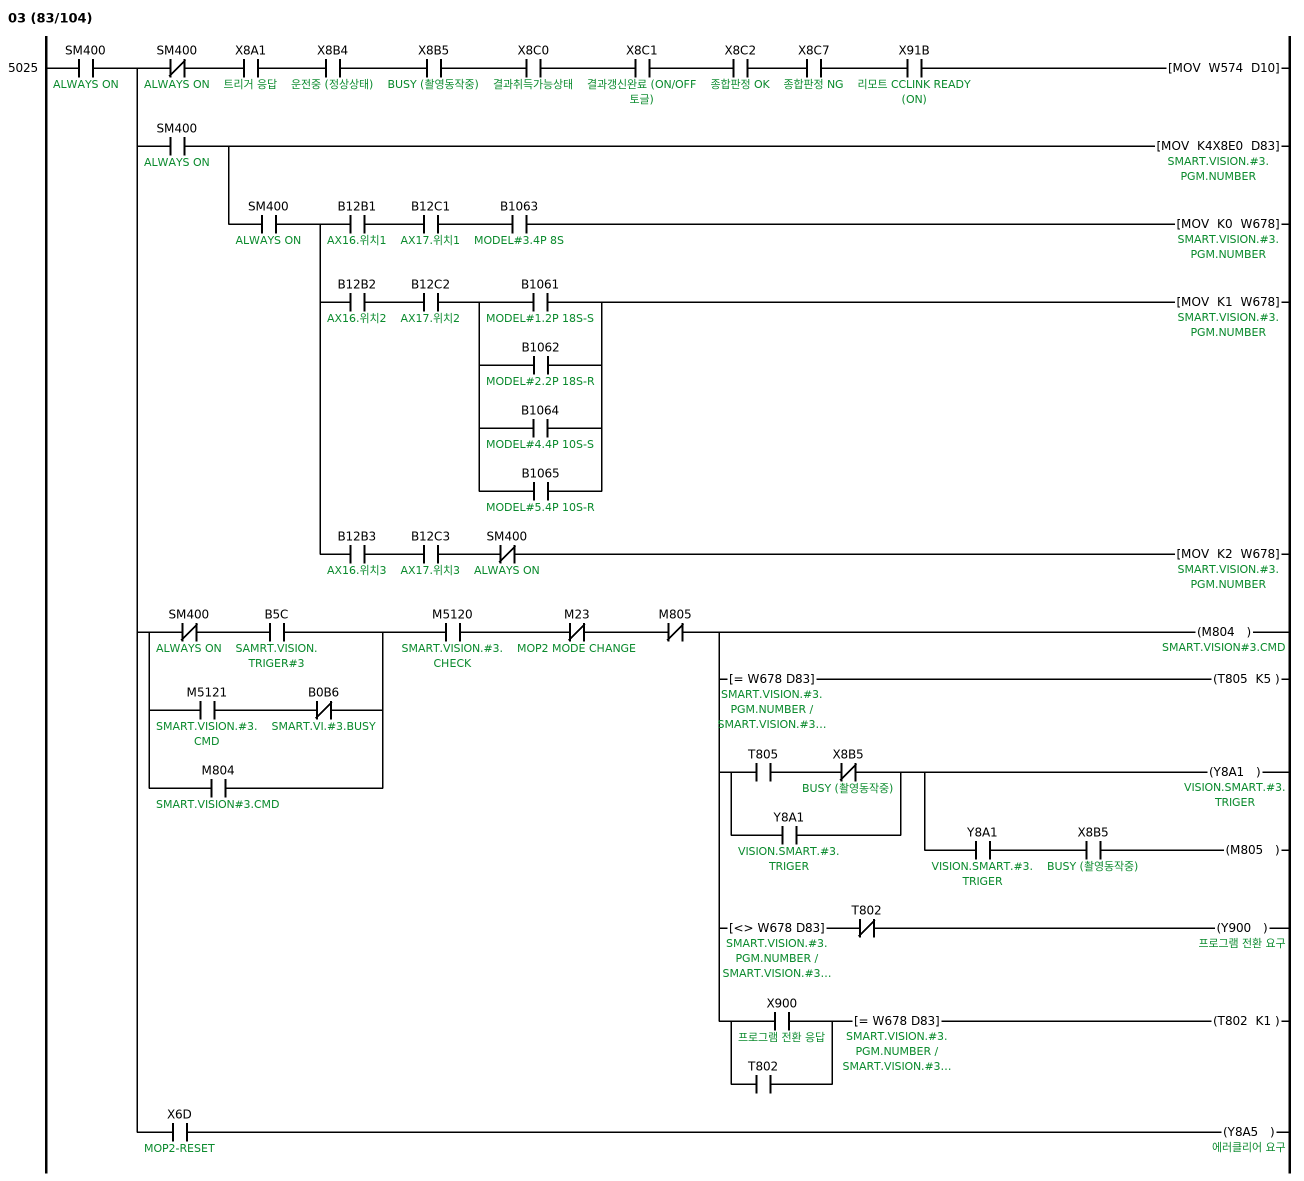
5025  LD      SM400  ; ALWAYS ON
      MPS
      ANI     SM400  ; ALWAYS ON
      AND     X8A1  ; 트리거 응답
      AND     X8B4  ; 운전중 (정상상태)
      AND     X8B5  ; BUSY (촬영동작중)
      AND     X8C0  ; 결과취득가능상태
      AND     X8C1  ; 결과갱신완료 (ON/OFF 토글)
      AND     X8C2  ; 종합판정 OK
      AND     X8C7  ; 종합판정 NG
      AND     X91B  ; 리모트 CCLINK READY (ON)
      MOV     W574 D10
      MRD
      AND     SM400  ; ALWAYS ON
      MOV     K4X8E0 D83  ; 프로그램번호 (BIT 0) / SMART.VISION.#3.PGM.NUMBER
      AND     SM400  ; ALWAYS ON
      MPS
      AND     B12B1  ; AX16.위치1
      AND     B12C1  ; AX17.위치1
      AND     B1063  ; MODEL#3.4P 8S
      MOV     K0 W678  ; SMART.VISION.#3.PGM.NUMBER
      MRD
      AND     B12B2  ; AX16.위치2
      AND     B12C2  ; AX17.위치2
      LD      B1061  ; MODEL#1.2P 18S-S
      OR      B1062  ; MODEL#2.2P 18S-R
      OR      B1064  ; MODEL#4.4P 10S-S
      OR      B1065  ; MODEL#5.4P 10S-R
      ANB
      MOV     K1 W678
      MPP
      AND     B12B3  ; AX16.위치3
      AND     B12C3  ; AX17.위치3
      ANI     SM400  ; ALWAYS ON
      MOV     K2 W678
      MRD
      LDI     SM400  ; ALWAYS ON
      AND     B5C  ; SAMRT.VISION.TRIGER#3
      LD      M5121  ; SMART.VISION.#3.CMD
      ANI     B0B6  ; SMART.VI.#3.BUSY
      ORB
      OR      M804  ; SMART.VISION#3.CMD
      ANB
      AND     M5120  ; SMART.VISION.#3.CHECK
      ANI     M23  ; MOP2 MODE CHANGE
      ANI     M805
      OUT     M804  ; SMART.VISION#3.CMD
      MPS
      AND=    W678 D83  ; SMART.VISION.#3.PGM.NUMBER / SMART.VISION.#3.PGM.NUMBER
      OUT     T805 K5
      MRD
      LD      T805
      ANI     X8B5  ; BUSY (촬영동작중)
      OR      Y8A1  ; VISION.SMART.#3.TRIGER
      ANB
      OUT     Y8A1  ; VISION.SMART.#3.TRIGER
      AND     Y8A1  ; VISION.SMART.#3.TRIGER
      AND     X8B5  ; BUSY (촬영동작중)
      OUT     M805
      MRD
      AND<>   W678 D83  ; SMART.VISION.#3.PGM.NUMBER / SMART.VISION.#3.PGM.NUMBER
      ANI     T802
      OUT     Y900  ; 프로그램 전환 요구
      MPP
      LD      X900  ; 프로그램 전환 응답
      OR      T802
      ANB
      AND=    W678 D83  ; SMART.VISION.#3.PGM.NUMBER / SMART.VISION.#3.PGM.NUMBER
      OUT     T802 K1
      MPP
      AND     X6D  ; MOP2-RESET
      OUT     Y8A5  ; 에러클리어 요구
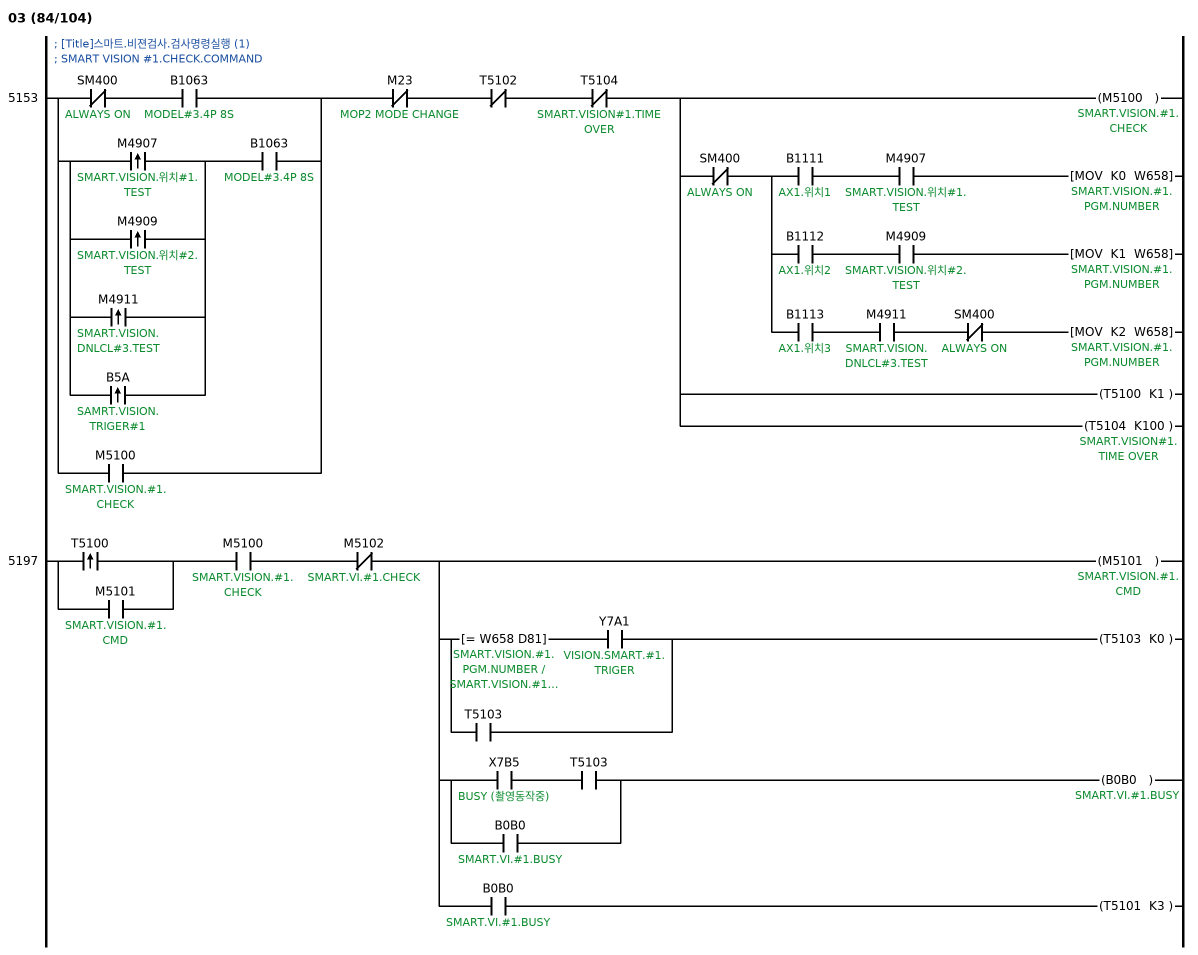
; [Title]스마트.비젼검사.검사명령실행 (1)
; SMART VISION #1.CHECK.COMMAND
5153  LDI     SM400  ; ALWAYS ON
      AND     B1063  ; MODEL#3.4P 8S
      LDP     M4907  ; SMART.VISION.위치#1.TEST
      ORP     M4909  ; SMART.VISION.위치#2.TEST
      ORP     M4911  ; SMART.VISION.DNLCL#3.TEST
      ORP     B5A  ; SAMRT.VISION.TRIGER#1
      AND     B1063  ; MODEL#3.4P 8S
      ORB
      OR      M5100  ; SMART.VISION.#1.CHECK
      ANI     M23  ; MOP2 MODE CHANGE
      ANI     T5102
      ANI     T5104  ; SMART.VISION#1.TIME OVER
      OUT     M5100  ; SMART.VISION.#1.CHECK
      MPS
      ANI     SM400  ; ALWAYS ON
      MPS
      AND     B1111  ; AX1.위치1
      AND     M4907  ; SMART.VISION.위치#1.TEST
      MOV     K0 W658
      MRD
      AND     B1112  ; AX1.위치2
      AND     M4909  ; SMART.VISION.위치#2.TEST
      MOV     K1 W658
      MPP
      AND     B1113  ; AX1.위치3
      AND     M4911  ; SMART.VISION.DNLCL#3.TEST
      ANI     SM400  ; ALWAYS ON
      MOV     K2 W658
      MPP
      OUT     T5100 K1
      OUT     T5104 K100  ; SMART.VISION#1.TIME OVER
5197  LDP     T5100
      OR      M5101  ; SMART.VISION.#1.CMD
      AND     M5100  ; SMART.VISION.#1.CHECK
      ANI     M5102  ; SMART.VI.#1.CHECK
      OUT     M5101  ; SMART.VISION.#1.CMD
      MPS
      LD=     W658 D81  ; SMART.VISION.#1.PGM.NUMBER / SMART.VISION.#1.PGM.NUMBER
      AND     Y7A1  ; VISION.SMART.#1.TRIGER
      OR      T5103
      ANB
      OUT     T5103 K0
      MRD
      LD      X7B5  ; BUSY (촬영동작중)
      AND     T5103
      OR      B0B0  ; SMART.VI.#1.BUSY
      ANB
      OUT     B0B0  ; SMART.VI.#1.BUSY
      MPP
      AND     B0B0  ; SMART.VI.#1.BUSY
      OUT     T5101 K3
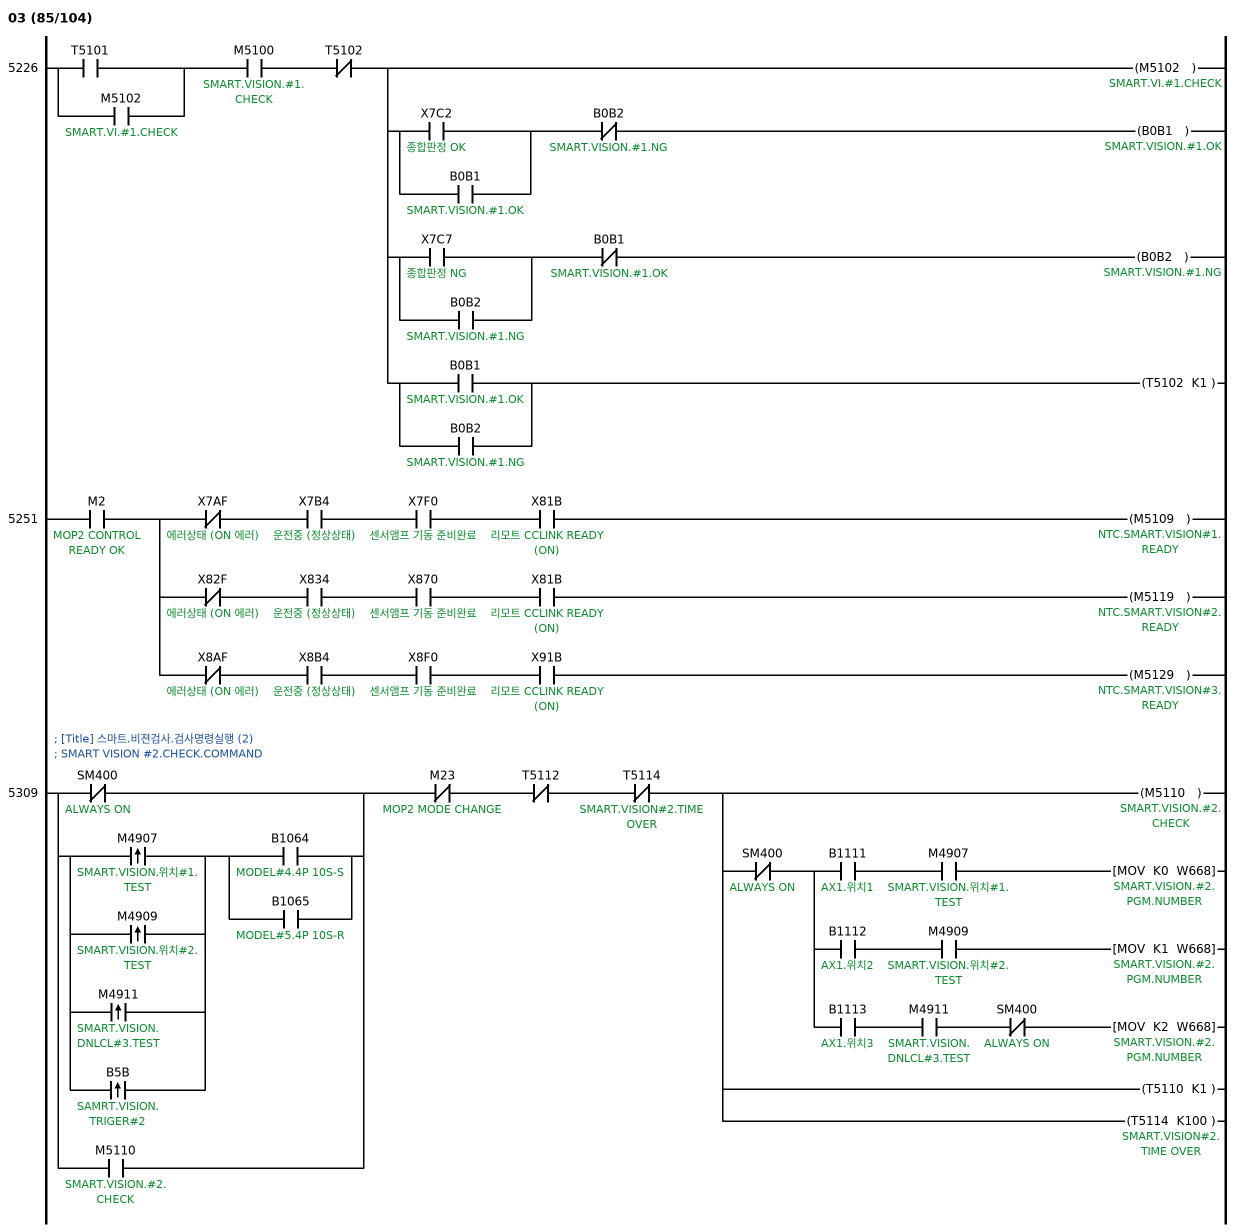
5226  LD      T5101
      OR      M5102  ; SMART.VI.#1.CHECK
      AND     M5100  ; SMART.VISION.#1.CHECK
      ANI     T5102
      OUT     M5102  ; SMART.VI.#1.CHECK
      MPS
      LD      X7C2  ; 종합판정 OK
      OR      B0B1  ; SMART.VISION.#1.OK
      ANB
      ANI     B0B2  ; SMART.VISION.#1.NG
      OUT     B0B1  ; SMART.VISION.#1.OK
      MRD
      LD      X7C7  ; 종합판정 NG
      OR      B0B2  ; SMART.VISION.#1.NG
      ANB
      ANI     B0B1  ; SMART.VISION.#1.OK
      OUT     B0B2  ; SMART.VISION.#1.NG
      MPP
      LD      B0B1  ; SMART.VISION.#1.OK
      OR      B0B2  ; SMART.VISION.#1.NG
      ANB
      OUT     T5102 K1
5251  LD      M2  ; MOP2 CONTROL READY OK
      MPS
      ANI     X7AF  ; 에러상태 (ON 에러)
      AND     X7B4  ; 운전중 (정상상태)
      AND     X7F0  ; 센서앰프 기동 준비완료
      AND     X81B  ; 리모트 CCLINK READY (ON)
      OUT     M5109  ; NTC.SMART.VISION#1.READY
      MRD
      ANI     X82F  ; 에러상태 (ON 에러)
      AND     X834  ; 운전중 (정상상태)
      AND     X870  ; 센서앰프 기동 준비완료
      AND     X81B  ; 리모트 CCLINK READY (ON)
      OUT     M5119  ; NTC.SMART.VISION#2.READY
      MPP
      ANI     X8AF  ; 에러상태 (ON 에러)
      AND     X8B4  ; 운전중 (정상상태)
      AND     X8F0  ; 센서앰프 기동 준비완료
      AND     X91B  ; 리모트 CCLINK READY (ON)
      OUT     M5129  ; NTC.SMART.VISION#3.READY
; [Title] 스마트.비젼검사.검사명령실행 (2)
; SMART VISION #2.CHECK.COMMAND
5309  LDI     SM400  ; ALWAYS ON
      LDP     M4907  ; SMART.VISION.위치#1.TEST
      ORP     M4909  ; SMART.VISION.위치#2.TEST
      ORP     M4911  ; SMART.VISION.DNLCL#3.TEST
      ORP     B5B  ; SAMRT.VISION.TRIGER#2
      LD      B1064  ; MODEL#4.4P 10S-S
      OR      B1065  ; MODEL#5.4P 10S-R
      ANB
      ORB
      OR      M5110  ; SMART.VISION.#2.CHECK
      ANI     M23  ; MOP2 MODE CHANGE
      ANI     T5112
      ANI     T5114  ; SMART.VISION#2.TIME OVER
      OUT     M5110  ; SMART.VISION.#2.CHECK
      MPS
      ANI     SM400  ; ALWAYS ON
      MPS
      AND     B1111  ; AX1.위치1
      AND     M4907  ; SMART.VISION.위치#1.TEST
      MOV     K0 W668
      MRD
      AND     B1112  ; AX1.위치2
      AND     M4909  ; SMART.VISION.위치#2.TEST
      MOV     K1 W668
      MPP
      AND     B1113  ; AX1.위치3
      AND     M4911  ; SMART.VISION.DNLCL#3.TEST
      ANI     SM400  ; ALWAYS ON
      MOV     K2 W668
      MPP
      OUT     T5110 K1
      OUT     T5114 K100  ; SMART.VISION#2.TIME OVER
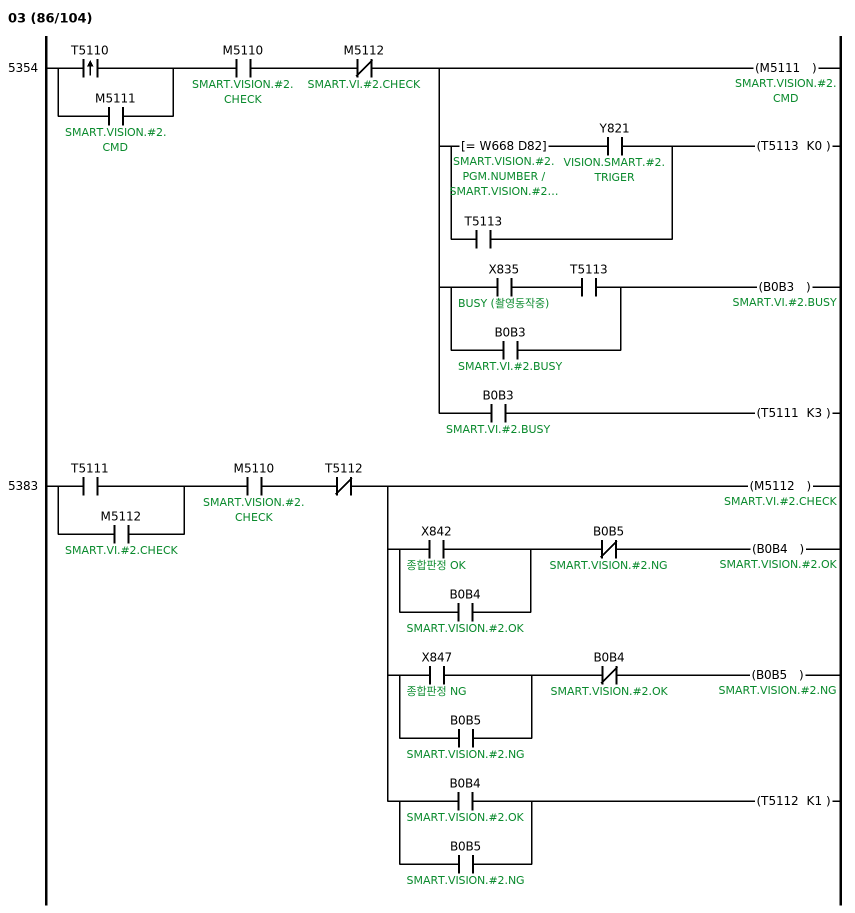
5354  LDP     T5110
      OR      M5111  ; SMART.VISION.#2.CMD
      AND     M5110  ; SMART.VISION.#2.CHECK
      ANI     M5112  ; SMART.VI.#2.CHECK
      OUT     M5111  ; SMART.VISION.#2.CMD
      MPS
      LD=     W668 D82  ; SMART.VISION.#2.PGM.NUMBER / SMART.VISION.#2.PGM.NUMBER
      AND     Y821  ; VISION.SMART.#2.TRIGER
      OR      T5113
      ANB
      OUT     T5113 K0
      MRD
      LD      X835  ; BUSY (촬영동작중)
      AND     T5113
      OR      B0B3  ; SMART.VI.#2.BUSY
      ANB
      OUT     B0B3  ; SMART.VI.#2.BUSY
      MPP
      AND     B0B3  ; SMART.VI.#2.BUSY
      OUT     T5111 K3
5383  LD      T5111
      OR      M5112  ; SMART.VI.#2.CHECK
      AND     M5110  ; SMART.VISION.#2.CHECK
      ANI     T5112
      OUT     M5112  ; SMART.VI.#2.CHECK
      MPS
      LD      X842  ; 종합판정 OK
      OR      B0B4  ; SMART.VISION.#2.OK
      ANB
      ANI     B0B5  ; SMART.VISION.#2.NG
      OUT     B0B4  ; SMART.VISION.#2.OK
      MRD
      LD      X847  ; 종합판정 NG
      OR      B0B5  ; SMART.VISION.#2.NG
      ANB
      ANI     B0B4  ; SMART.VISION.#2.OK
      OUT     B0B5  ; SMART.VISION.#2.NG
      MPP
      LD      B0B4  ; SMART.VISION.#2.OK
      OR      B0B5  ; SMART.VISION.#2.NG
      ANB
      OUT     T5112 K1
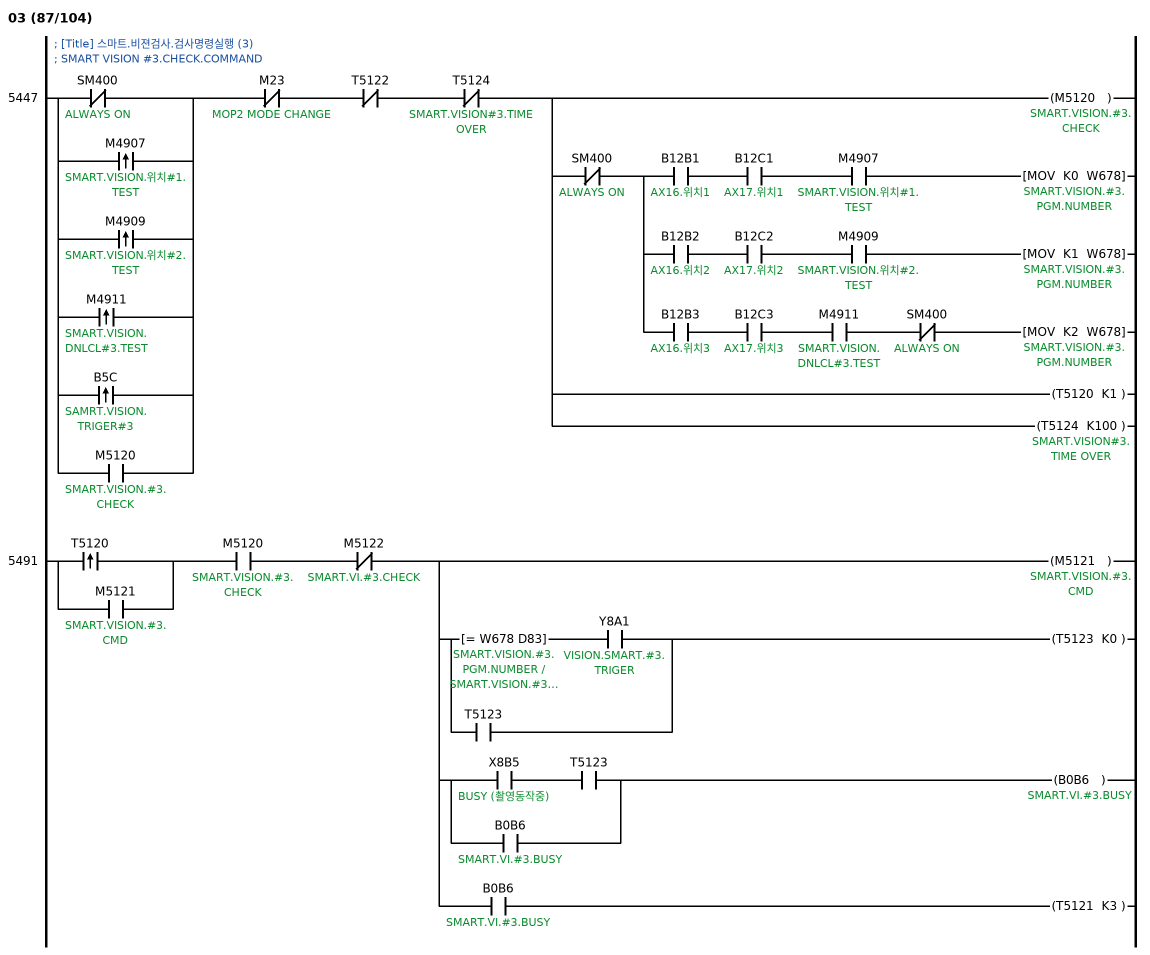
; [Title] 스마트.비젼검사.검사명령실행 (3)
; SMART VISION #3.CHECK.COMMAND
5447  LDI     SM400  ; ALWAYS ON
      ORP     M4907  ; SMART.VISION.위치#1.TEST
      ORP     M4909  ; SMART.VISION.위치#2.TEST
      ORP     M4911  ; SMART.VISION.DNLCL#3.TEST
      ORP     B5C  ; SAMRT.VISION.TRIGER#3
      OR      M5120  ; SMART.VISION.#3.CHECK
      ANI     M23  ; MOP2 MODE CHANGE
      ANI     T5122
      ANI     T5124  ; SMART.VISION#3.TIME OVER
      OUT     M5120  ; SMART.VISION.#3.CHECK
      MPS
      ANI     SM400  ; ALWAYS ON
      MPS
      AND     B12B1  ; AX16.위치1
      AND     B12C1  ; AX17.위치1
      AND     M4907  ; SMART.VISION.위치#1.TEST
      MOV     K0 W678
      MRD
      AND     B12B2  ; AX16.위치2
      AND     B12C2  ; AX17.위치2
      AND     M4909  ; SMART.VISION.위치#2.TEST
      MOV     K1 W678
      MPP
      AND     B12B3  ; AX16.위치3
      AND     B12C3  ; AX17.위치3
      AND     M4911  ; SMART.VISION.DNLCL#3.TEST
      ANI     SM400  ; ALWAYS ON
      MOV     K2 W678
      MPP
      OUT     T5120 K1
      OUT     T5124 K100  ; SMART.VISION#3.TIME OVER
5491  LDP     T5120
      OR      M5121  ; SMART.VISION.#3.CMD
      AND     M5120  ; SMART.VISION.#3.CHECK
      ANI     M5122  ; SMART.VI.#3.CHECK
      OUT     M5121  ; SMART.VISION.#3.CMD
      MPS
      LD=     W678 D83  ; SMART.VISION.#3.PGM.NUMBER / SMART.VISION.#3.PGM.NUMBER
      AND     Y8A1  ; VISION.SMART.#3.TRIGER
      OR      T5123
      ANB
      OUT     T5123 K0
      MRD
      LD      X8B5  ; BUSY (촬영동작중)
      AND     T5123
      OR      B0B6  ; SMART.VI.#3.BUSY
      ANB
      OUT     B0B6  ; SMART.VI.#3.BUSY
      MPP
      AND     B0B6  ; SMART.VI.#3.BUSY
      OUT     T5121 K3
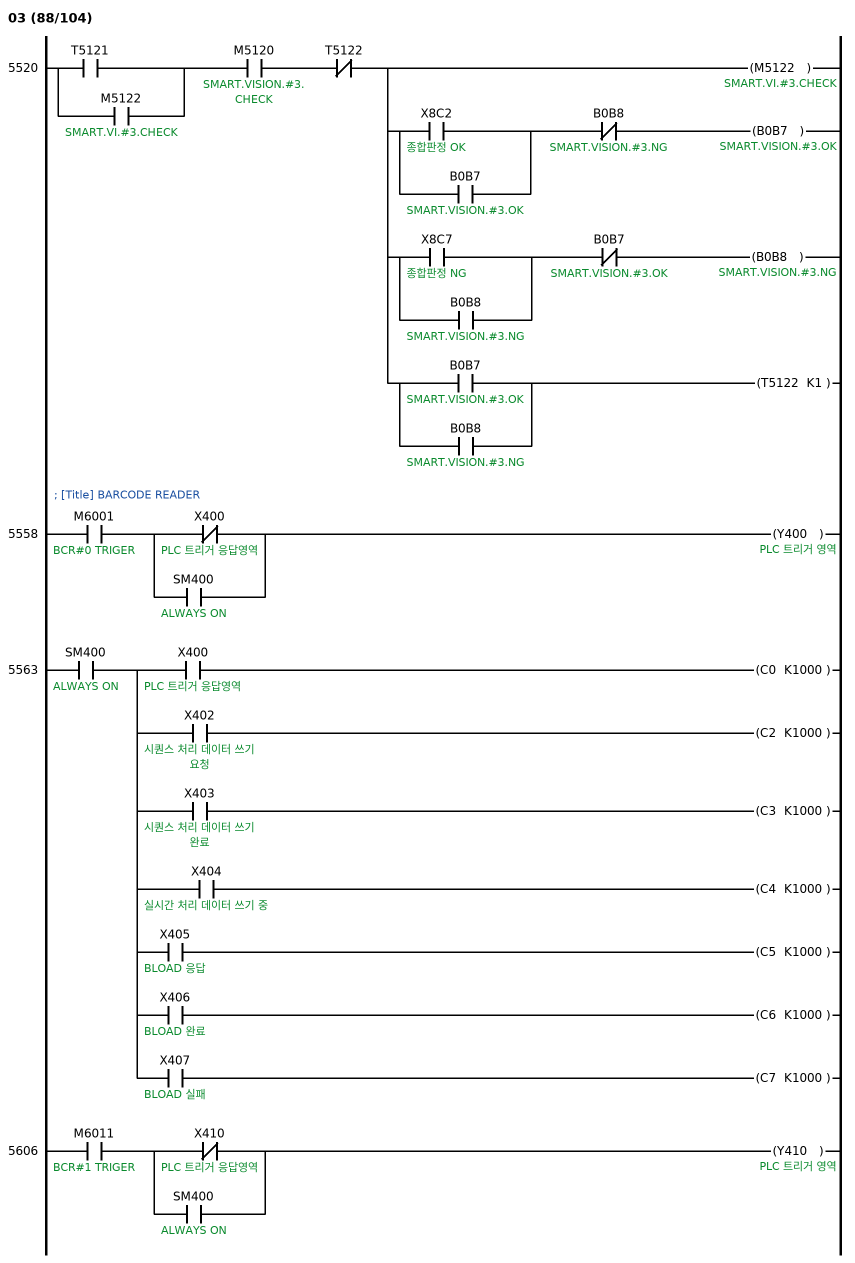
5520  LD      T5121
      OR      M5122  ; SMART.VI.#3.CHECK
      AND     M5120  ; SMART.VISION.#3.CHECK
      ANI     T5122
      OUT     M5122  ; SMART.VI.#3.CHECK
      MPS
      LD      X8C2  ; 종합판정 OK
      OR      B0B7  ; SMART.VISION.#3.OK
      ANB
      ANI     B0B8  ; SMART.VISION.#3.NG
      OUT     B0B7  ; SMART.VISION.#3.OK
      MRD
      LD      X8C7  ; 종합판정 NG
      OR      B0B8  ; SMART.VISION.#3.NG
      ANB
      ANI     B0B7  ; SMART.VISION.#3.OK
      OUT     B0B8  ; SMART.VISION.#3.NG
      MPP
      LD      B0B7  ; SMART.VISION.#3.OK
      OR      B0B8  ; SMART.VISION.#3.NG
      ANB
      OUT     T5122 K1
; [Title] BARCODE READER
5558  LD      M6001  ; BCR#0 TRIGER
      LDI     X400  ; PLC 트리거 응답영역
      OR      SM400  ; ALWAYS ON
      ANB
      OUT     Y400  ; PLC 트리거 영역
5563  LD      SM400  ; ALWAYS ON
      MPS
      AND     X400  ; PLC 트리거 응답영역
      OUT     C0 K1000
      MRD
      AND     X402  ; 시퀀스 처리 데이터 쓰기 요청
      OUT     C2 K1000
      MRD
      AND     X403  ; 시퀀스 처리 데이터 쓰기 완료
      OUT     C3 K1000
      MRD
      AND     X404  ; 실시간 처리 데이터 쓰기 중
      OUT     C4 K1000
      MRD
      AND     X405  ; BLOAD 응답
      OUT     C5 K1000
      MRD
      AND     X406  ; BLOAD 완료
      OUT     C6 K1000
      MPP
      AND     X407  ; BLOAD 실패
      OUT     C7 K1000
5606  LD      M6011  ; BCR#1 TRIGER
      LDI     X410  ; PLC 트리거 응답영역
      OR      SM400  ; ALWAYS ON
      ANB
      OUT     Y410  ; PLC 트리거 영역
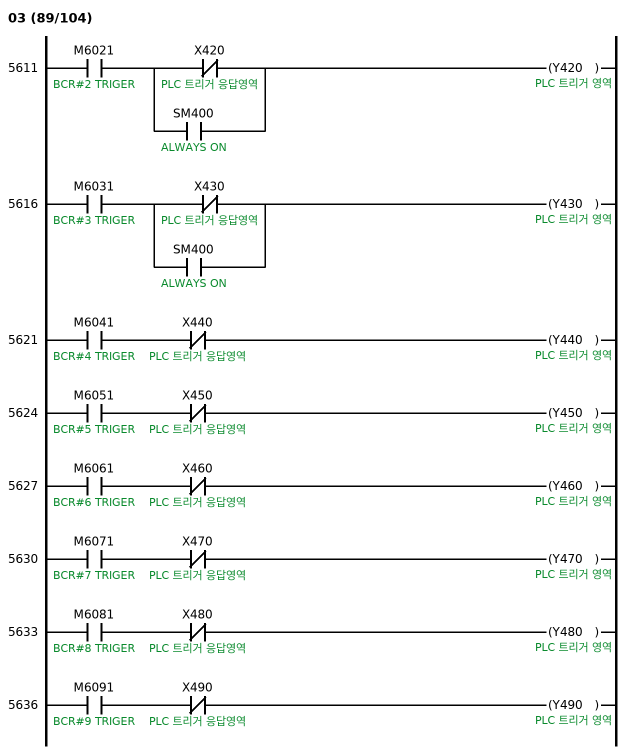
5611  LD      M6021  ; BCR#2 TRIGER
      LDI     X420  ; PLC 트리거 응답영역
      OR      SM400  ; ALWAYS ON
      ANB
      OUT     Y420  ; PLC 트리거 영역
5616  LD      M6031  ; BCR#3 TRIGER
      LDI     X430  ; PLC 트리거 응답영역
      OR      SM400  ; ALWAYS ON
      ANB
      OUT     Y430  ; PLC 트리거 영역
5621  LD      M6041  ; BCR#4 TRIGER
      ANI     X440  ; PLC 트리거 응답영역
      OUT     Y440  ; PLC 트리거 영역
5624  LD      M6051  ; BCR#5 TRIGER
      ANI     X450  ; PLC 트리거 응답영역
      OUT     Y450  ; PLC 트리거 영역
5627  LD      M6061  ; BCR#6 TRIGER
      ANI     X460  ; PLC 트리거 응답영역
      OUT     Y460  ; PLC 트리거 영역
5630  LD      M6071  ; BCR#7 TRIGER
      ANI     X470  ; PLC 트리거 응답영역
      OUT     Y470  ; PLC 트리거 영역
5633  LD      M6081  ; BCR#8 TRIGER
      ANI     X480  ; PLC 트리거 응답영역
      OUT     Y480  ; PLC 트리거 영역
5636  LD      M6091  ; BCR#9 TRIGER
      ANI     X490  ; PLC 트리거 응답영역
      OUT     Y490  ; PLC 트리거 영역
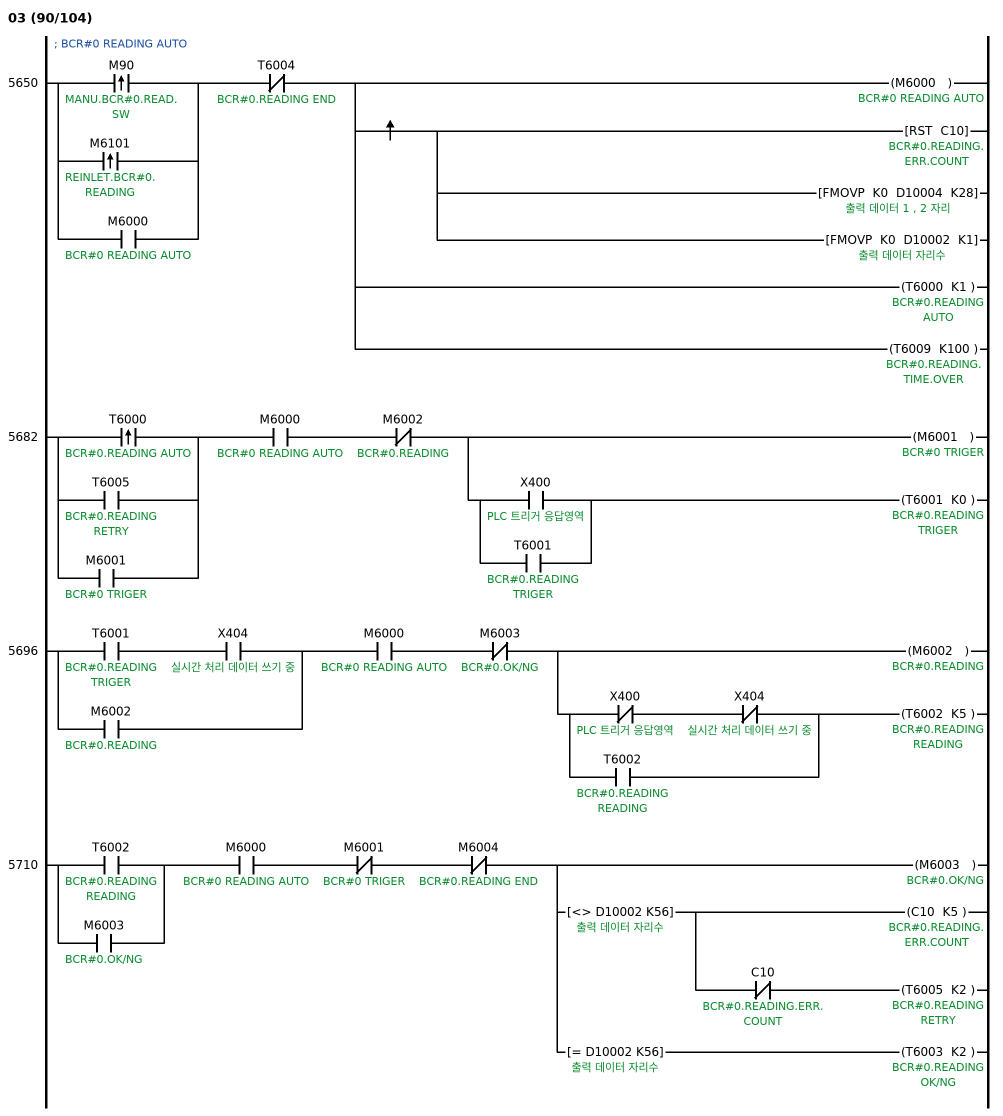
; BCR#0 READING AUTO
5650  LDP     M90  ; MANU.BCR#0.READ.SW
      ORP     M6101  ; REINLET.BCR#0.READING
      OR      M6000  ; BCR#0 READING AUTO
      ANI     T6004  ; BCR#0.READING END
      OUT     M6000  ; BCR#0 READING AUTO
      MPS
      MEP
      RST     C10  ; BCR#0.READING.ERR.COUNT
      FMOVP   K0 D10004 K28  ; 출력 데이터 1 , 2 자리
      FMOVP   K0 D10002 K1  ; 출력 데이터 자리수
      MPP
      OUT     T6000 K1  ; BCR#0.READING AUTO
      OUT     T6009 K100  ; BCR#0.READING.TIME.OVER
5682  LDP     T6000  ; BCR#0.READING AUTO
      OR      T6005  ; BCR#0.READING RETRY
      OR      M6001  ; BCR#0 TRIGER
      AND     M6000  ; BCR#0 READING AUTO
      ANI     M6002  ; BCR#0.READING
      OUT     M6001  ; BCR#0 TRIGER
      LD      X400  ; PLC 트리거 응답영역
      OR      T6001  ; BCR#0.READING TRIGER
      ANB
      OUT     T6001 K0  ; BCR#0.READING TRIGER
5696  LD      T6001  ; BCR#0.READING TRIGER
      AND     X404  ; 실시간 처리 데이터 쓰기 중
      OR      M6002  ; BCR#0.READING
      AND     M6000  ; BCR#0 READING AUTO
      ANI     M6003  ; BCR#0.OK/NG
      OUT     M6002  ; BCR#0.READING
      LDI     X400  ; PLC 트리거 응답영역
      ANI     X404  ; 실시간 처리 데이터 쓰기 중
      OR      T6002  ; BCR#0.READING READING
      ANB
      OUT     T6002 K5  ; BCR#0.READING READING
5710  LD      T6002  ; BCR#0.READING READING
      OR      M6003  ; BCR#0.OK/NG
      AND     M6000  ; BCR#0 READING AUTO
      ANI     M6001  ; BCR#0 TRIGER
      ANI     M6004  ; BCR#0.READING END
      OUT     M6003  ; BCR#0.OK/NG
      MPS
      AND<>   D10002 K56  ; 출력 데이터 자리수
      OUT     C10 K5  ; BCR#0.READING.ERR.COUNT
      ANI     C10  ; BCR#0.READING.ERR.COUNT
      OUT     T6005 K2  ; BCR#0.READING RETRY
      MPP
      AND=    D10002 K56  ; 출력 데이터 자리수
      OUT     T6003 K2  ; BCR#0.READING OK/NG
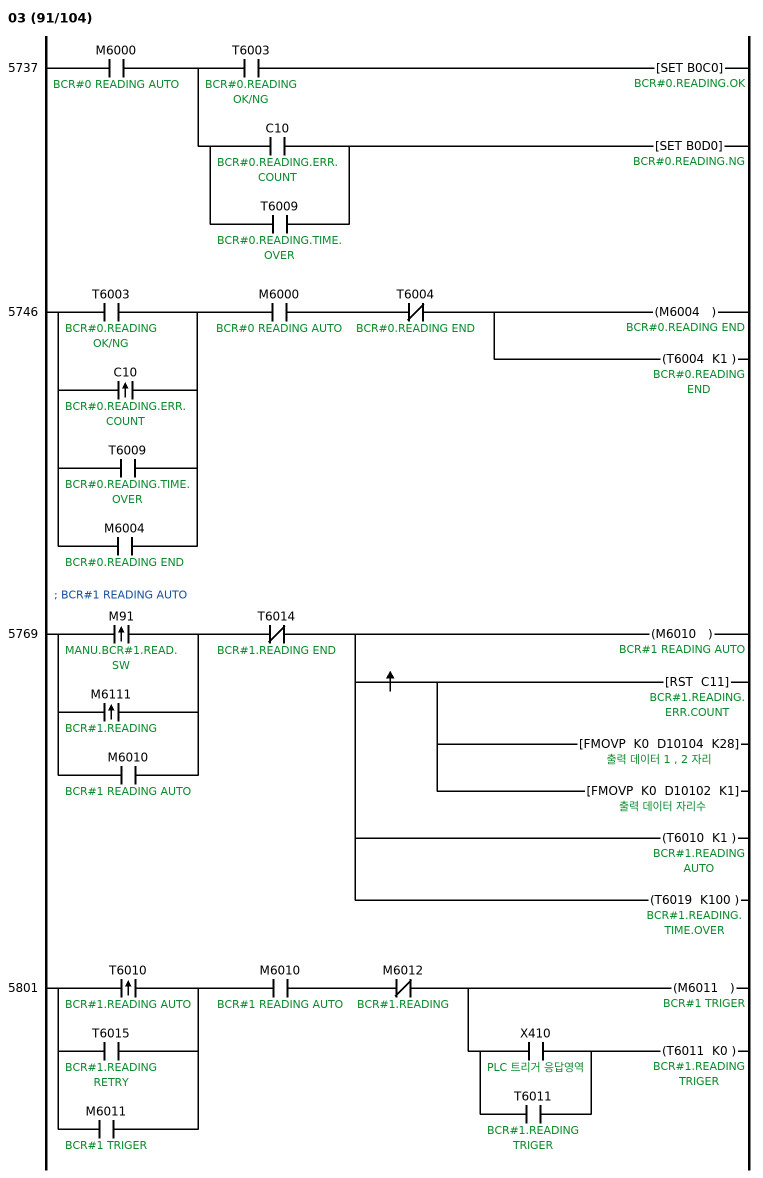
5737  LD      M6000  ; BCR#0 READING AUTO
      MPS
      AND     T6003  ; BCR#0.READING OK/NG
      SET     B0C0  ; BCR#0.READING.OK
      MPP
      LD      C10  ; BCR#0.READING.ERR.COUNT
      OR      T6009  ; BCR#0.READING.TIME.OVER
      ANB
      SET     B0D0  ; BCR#0.READING.NG
5746  LD      T6003  ; BCR#0.READING OK/NG
      ORP     C10  ; BCR#0.READING.ERR.COUNT
      OR      T6009  ; BCR#0.READING.TIME.OVER
      OR      M6004  ; BCR#0.READING END
      AND     M6000  ; BCR#0 READING AUTO
      ANI     T6004  ; BCR#0.READING END
      OUT     M6004  ; BCR#0.READING END
      OUT     T6004 K1  ; BCR#0.READING END
; BCR#1 READING AUTO
5769  LDP     M91  ; MANU.BCR#1.READ.SW
      ORP     M6111  ; BCR#1.READING
      OR      M6010  ; BCR#1 READING AUTO
      ANI     T6014  ; BCR#1.READING END
      OUT     M6010  ; BCR#1 READING AUTO
      MPS
      MEP
      RST     C11  ; BCR#1.READING.ERR.COUNT
      FMOVP   K0 D10104 K28  ; 출력 데이터 1 , 2 자리
      FMOVP   K0 D10102 K1  ; 출력 데이터 자리수
      MPP
      OUT     T6010 K1  ; BCR#1.READING AUTO
      OUT     T6019 K100  ; BCR#1.READING.TIME.OVER
5801  LDP     T6010  ; BCR#1.READING AUTO
      OR      T6015  ; BCR#1.READING RETRY
      OR      M6011  ; BCR#1 TRIGER
      AND     M6010  ; BCR#1 READING AUTO
      ANI     M6012  ; BCR#1.READING
      OUT     M6011  ; BCR#1 TRIGER
      LD      X410  ; PLC 트리거 응답영역
      OR      T6011  ; BCR#1.READING TRIGER
      ANB
      OUT     T6011 K0  ; BCR#1.READING TRIGER
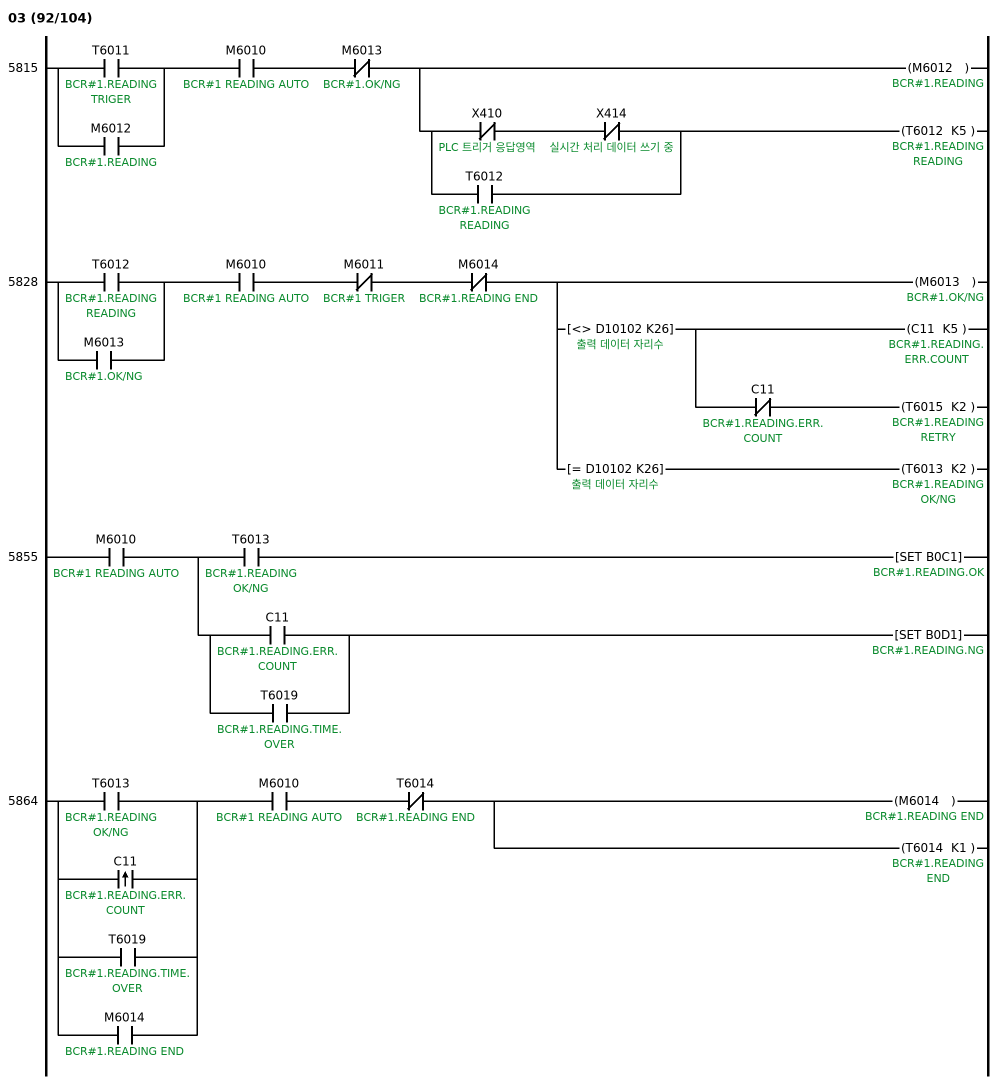
5815  LD      T6011  ; BCR#1.READING TRIGER
      OR      M6012  ; BCR#1.READING
      AND     M6010  ; BCR#1 READING AUTO
      ANI     M6013  ; BCR#1.OK/NG
      OUT     M6012  ; BCR#1.READING
      LDI     X410  ; PLC 트리거 응답영역
      ANI     X414  ; 실시간 처리 데이터 쓰기 중
      OR      T6012  ; BCR#1.READING READING
      ANB
      OUT     T6012 K5  ; BCR#1.READING READING
5828  LD      T6012  ; BCR#1.READING READING
      OR      M6013  ; BCR#1.OK/NG
      AND     M6010  ; BCR#1 READING AUTO
      ANI     M6011  ; BCR#1 TRIGER
      ANI     M6014  ; BCR#1.READING END
      OUT     M6013  ; BCR#1.OK/NG
      MPS
      AND<>   D10102 K26  ; 출력 데이터 자리수
      OUT     C11 K5  ; BCR#1.READING.ERR.COUNT
      ANI     C11  ; BCR#1.READING.ERR.COUNT
      OUT     T6015 K2  ; BCR#1.READING RETRY
      MPP
      AND=    D10102 K26  ; 출력 데이터 자리수
      OUT     T6013 K2  ; BCR#1.READING OK/NG
5855  LD      M6010  ; BCR#1 READING AUTO
      MPS
      AND     T6013  ; BCR#1.READING OK/NG
      SET     B0C1  ; BCR#1.READING.OK
      MPP
      LD      C11  ; BCR#1.READING.ERR.COUNT
      OR      T6019  ; BCR#1.READING.TIME.OVER
      ANB
      SET     B0D1  ; BCR#1.READING.NG
5864  LD      T6013  ; BCR#1.READING OK/NG
      ORP     C11  ; BCR#1.READING.ERR.COUNT
      OR      T6019  ; BCR#1.READING.TIME.OVER
      OR      M6014  ; BCR#1.READING END
      AND     M6010  ; BCR#1 READING AUTO
      ANI     T6014  ; BCR#1.READING END
      OUT     M6014  ; BCR#1.READING END
      OUT     T6014 K1  ; BCR#1.READING END
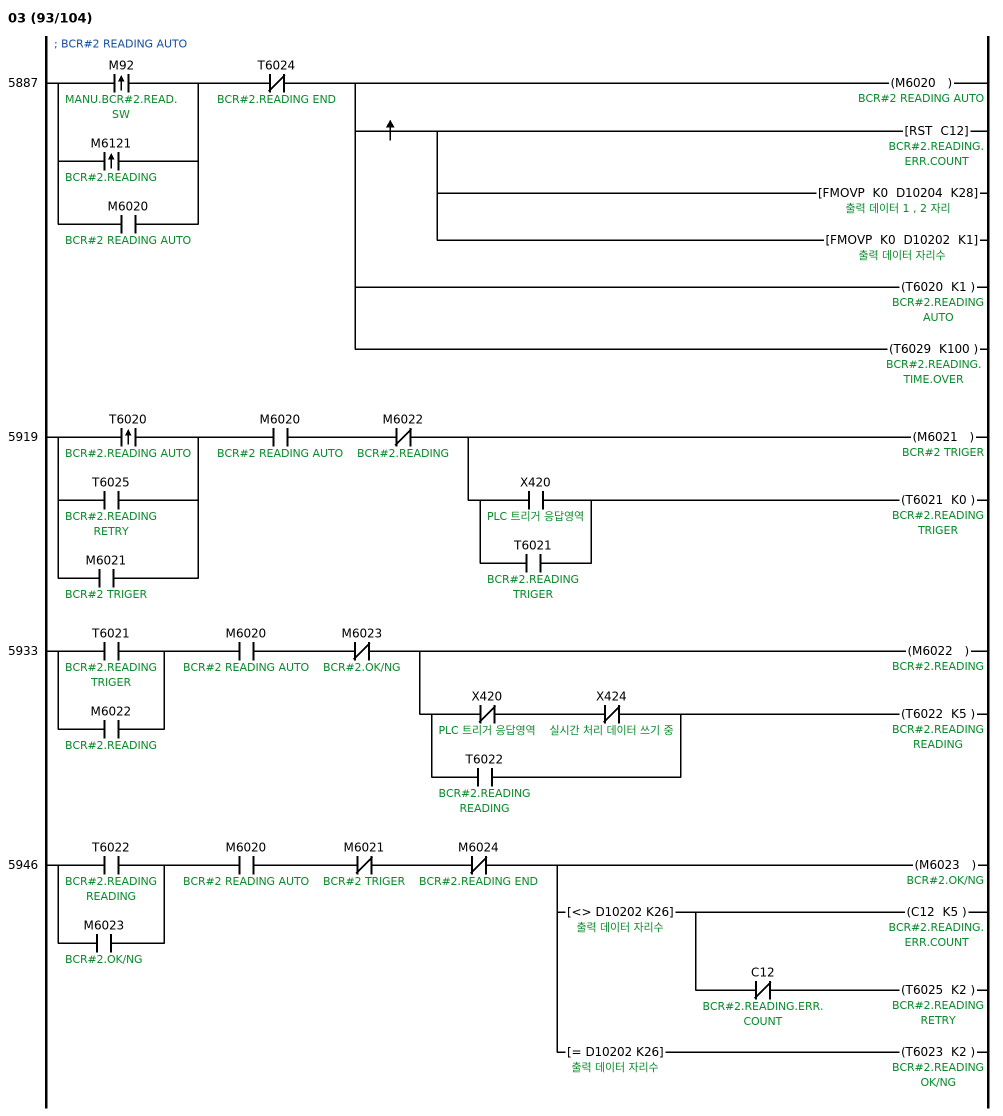
; BCR#2 READING AUTO
5887  LDP     M92  ; MANU.BCR#2.READ.SW
      ORP     M6121  ; BCR#2.READING
      OR      M6020  ; BCR#2 READING AUTO
      ANI     T6024  ; BCR#2.READING END
      OUT     M6020  ; BCR#2 READING AUTO
      MPS
      MEP
      RST     C12  ; BCR#2.READING.ERR.COUNT
      FMOVP   K0 D10204 K28  ; 출력 데이터 1 , 2 자리
      FMOVP   K0 D10202 K1  ; 출력 데이터 자리수
      MPP
      OUT     T6020 K1  ; BCR#2.READING AUTO
      OUT     T6029 K100  ; BCR#2.READING.TIME.OVER
5919  LDP     T6020  ; BCR#2.READING AUTO
      OR      T6025  ; BCR#2.READING RETRY
      OR      M6021  ; BCR#2 TRIGER
      AND     M6020  ; BCR#2 READING AUTO
      ANI     M6022  ; BCR#2.READING
      OUT     M6021  ; BCR#2 TRIGER
      LD      X420  ; PLC 트리거 응답영역
      OR      T6021  ; BCR#2.READING TRIGER
      ANB
      OUT     T6021 K0  ; BCR#2.READING TRIGER
5933  LD      T6021  ; BCR#2.READING TRIGER
      OR      M6022  ; BCR#2.READING
      AND     M6020  ; BCR#2 READING AUTO
      ANI     M6023  ; BCR#2.OK/NG
      OUT     M6022  ; BCR#2.READING
      LDI     X420  ; PLC 트리거 응답영역
      ANI     X424  ; 실시간 처리 데이터 쓰기 중
      OR      T6022  ; BCR#2.READING READING
      ANB
      OUT     T6022 K5  ; BCR#2.READING READING
5946  LD      T6022  ; BCR#2.READING READING
      OR      M6023  ; BCR#2.OK/NG
      AND     M6020  ; BCR#2 READING AUTO
      ANI     M6021  ; BCR#2 TRIGER
      ANI     M6024  ; BCR#2.READING END
      OUT     M6023  ; BCR#2.OK/NG
      MPS
      AND<>   D10202 K26  ; 출력 데이터 자리수
      OUT     C12 K5  ; BCR#2.READING.ERR.COUNT
      ANI     C12  ; BCR#2.READING.ERR.COUNT
      OUT     T6025 K2  ; BCR#2.READING RETRY
      MPP
      AND=    D10202 K26  ; 출력 데이터 자리수
      OUT     T6023 K2  ; BCR#2.READING OK/NG
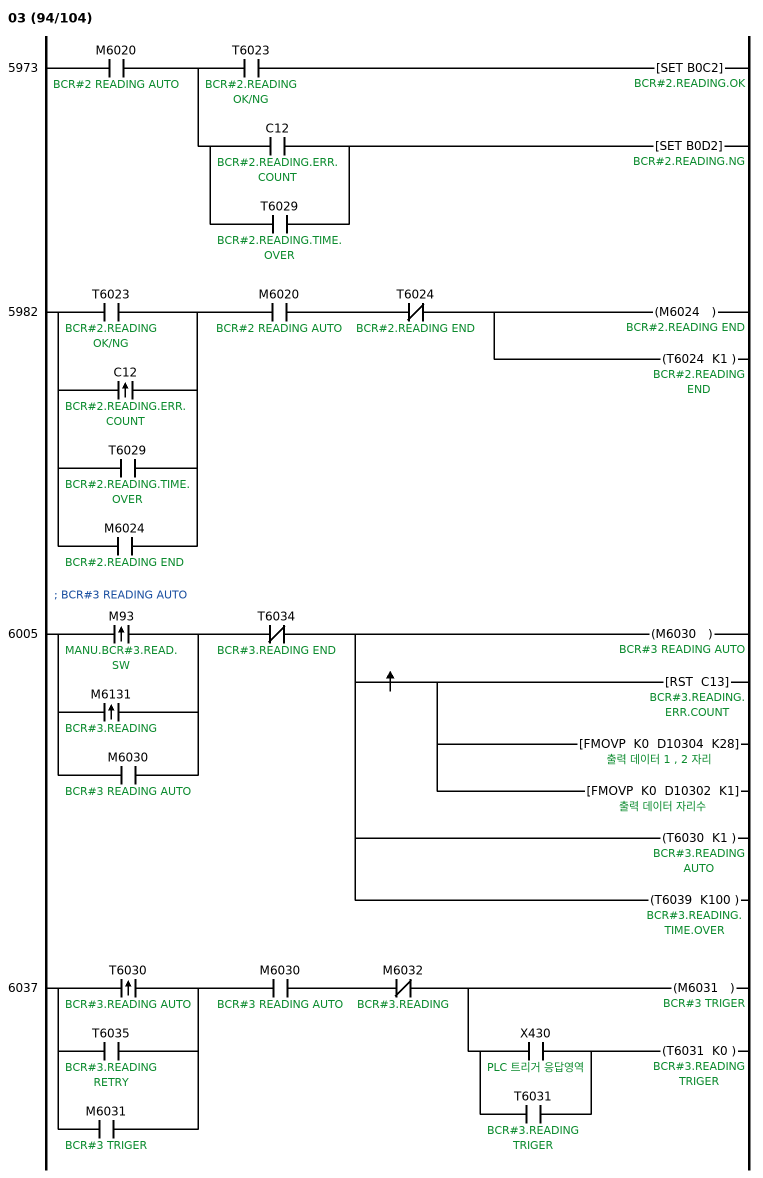
5973  LD      M6020  ; BCR#2 READING AUTO
      MPS
      AND     T6023  ; BCR#2.READING OK/NG
      SET     B0C2  ; BCR#2.READING.OK
      MPP
      LD      C12  ; BCR#2.READING.ERR.COUNT
      OR      T6029  ; BCR#2.READING.TIME.OVER
      ANB
      SET     B0D2  ; BCR#2.READING.NG
5982  LD      T6023  ; BCR#2.READING OK/NG
      ORP     C12  ; BCR#2.READING.ERR.COUNT
      OR      T6029  ; BCR#2.READING.TIME.OVER
      OR      M6024  ; BCR#2.READING END
      AND     M6020  ; BCR#2 READING AUTO
      ANI     T6024  ; BCR#2.READING END
      OUT     M6024  ; BCR#2.READING END
      OUT     T6024 K1  ; BCR#2.READING END
; BCR#3 READING AUTO
6005  LDP     M93  ; MANU.BCR#3.READ.SW
      ORP     M6131  ; BCR#3.READING
      OR      M6030  ; BCR#3 READING AUTO
      ANI     T6034  ; BCR#3.READING END
      OUT     M6030  ; BCR#3 READING AUTO
      MPS
      MEP
      RST     C13  ; BCR#3.READING.ERR.COUNT
      FMOVP   K0 D10304 K28  ; 출력 데이터 1 , 2 자리
      FMOVP   K0 D10302 K1  ; 출력 데이터 자리수
      MPP
      OUT     T6030 K1  ; BCR#3.READING AUTO
      OUT     T6039 K100  ; BCR#3.READING.TIME.OVER
6037  LDP     T6030  ; BCR#3.READING AUTO
      OR      T6035  ; BCR#3.READING RETRY
      OR      M6031  ; BCR#3 TRIGER
      AND     M6030  ; BCR#3 READING AUTO
      ANI     M6032  ; BCR#3.READING
      OUT     M6031  ; BCR#3 TRIGER
      LD      X430  ; PLC 트리거 응답영역
      OR      T6031  ; BCR#3.READING TRIGER
      ANB
      OUT     T6031 K0  ; BCR#3.READING TRIGER
